	X =  60.822  mm,	Y =   -346.772  mm,	Z =   -269.437  mm,
	W =  90.000 deg,	P =   0.000 deg,	R =   90.000 deg
};
P[82]{
   GP1:
	UF : 0, UT : 6,		CONFIG : 'N U T, 0, 0, 0',
	X =  61.497  mm,	Y =   -348.015  mm,	Z =   -269.167  mm,
	W =  90.000 deg,	P =   0.000 deg,	R =   90.000 deg
};
P[83]{
   GP1:
	UF : 0, UT : 6,		CONFIG : 'N U T, 0, 0, 0',
	X =  62.377  mm,	Y =   -349.588  mm,	Z =   -268.993  mm,
	W =  90.000 deg,	P =   0.000 deg,	R =   90.000 deg
};
P[84]{
   GP1:
	UF : 0, UT : 6,		CONFIG : 'N U T, 0, 0, 0',
	X =  62.802  mm,	Y =   -350.203  mm,	Z =   -269.422  mm,
	W =  90.000 deg,	P =   0.000 deg,	R =   90.000 deg
};
P[85]{
   GP1:
	UF : 0, UT : 6,		CONFIG : 'N U T, 0, 0, 0',
	X =  65.907  mm,	Y =   -355.659  mm,	Z =   -269.143  mm,
	W =  90.000 deg,	P =   0.000 deg,	R =   90.000 deg
};
P[86]{
   GP1:
	UF : 0, UT : 6,		CONFIG : 'N U T, 0, 0, 0',
	X =  66.444  mm,	Y =   -356.602  mm,	Z =   -269.105  mm,
	W =  90.000 deg,	P =   0.000 deg,	R =   90.000 deg
};
P[87]{
   GP1:
	UF : 0, UT : 6,		CONFIG : 'N U T, 0, 0, 0',
	X =  67.551  mm,	Y =   -358.541  mm,	Z =   -269.018  mm,
	W =  90.000 deg,	P =   0.000 deg,	R =   90.000 deg
};
P[88]{
   GP1:
	UF : 0, UT : 6,		CONFIG : 'N U T, 0, 0, 0',
	X =  68.086  mm,	Y =   -359.347  mm,	Z =   -269.445  mm,
	W =  90.000 deg,	P =   0.000 deg,	R =   90.000 deg
};
P[89]{
   GP1:
	UF : 0, UT : 6,		CONFIG : 'N U T, 0, 0, 0',
	X =  68.697  mm,	Y =   -360.426  mm,	Z =   -269.380  mm,
	W =  90.000 deg,	P =   0.000 deg,	R =   90.000 deg
};
P[90]{
   GP1:
	UF : 0, UT : 6,		CONFIG : 'N U T, 0, 0, 0',
	X =  69.791  mm,	Y =   -362.363  mm,	Z =   -269.223  mm,
	W =  90.000 deg,	P =   0.000 deg,	R =   90.000 deg
};
P[91]{
   GP1:
	UF : 0, UT : 6,		CONFIG : 'N U T, 0, 0, 0',
	X =  70.454  mm,	Y =   -363.448  mm,	Z =   -269.452  mm,
	W =  90.000 deg,	P =   0.000 deg,	R =   90.000 deg
};
P[92]{
   GP1:
	UF : 0, UT : 6,		CONFIG : 'N U T, 0, 0, 0',
	X =  71.652  mm,	Y =   -365.531  mm,	Z =   -269.420  mm,
	W =  90.000 deg,	P =   0.000 deg,	R =   90.000 deg
};
P[93]{
   GP1:
	UF : 0, UT : 6,		CONFIG : 'N U T, 0, 0, 0',
	X =  72.017  mm,	Y =   -366.190  mm,	Z =   -269.328  mm,
	W =  90.000 deg,	P =   0.000 deg,	R =   90.000 deg
};
P[94]{
   GP1:
	UF : 0, UT : 6,		CONFIG : 'N U T, 0, 0, 0',
	X =  73.518  mm,	Y =   -368.753  mm,	Z =   -269.459  mm,
	W =  90.000 deg,	P =   0.000 deg,	R =   90.000 deg
};
P[95]{
   GP1:
	UF : 0, UT : 6,		CONFIG : 'N U T, 0, 0, 0',
	X =  74.232  mm,	Y =   -370.046  mm,	Z =   -269.257  mm,
	W =  90.000 deg,	P =   0.000 deg,	R =   90.000 deg
};
P[96]{
   GP1:
	UF : 0, UT : 6,		CONFIG : 'N U T, 0, 0, 0',
	X =  75.118  mm,	Y =   -371.588  mm,	Z =   -269.233  mm,
	W =  90.000 deg,	P =   0.000 deg,	R =   90.000 deg
};
P[97]{
   GP1:
	UF : 0, UT : 6,		CONFIG : 'N U T, 0, 0, 0',
	X =  76.161  mm,	Y =   -373.400  mm,	Z =   -269.214  mm,
	W =  90.000 deg,	P =   0.000 deg,	R =   90.000 deg
};
P[98]{
   GP1:
	UF : 0, UT : 6,		CONFIG : 'N U T, 0, 0, 0',
	X =  76.622  mm,	Y =   -374.139  mm,	Z =   -269.425  mm,
	W =  90.000 deg,	P =   0.000 deg,	R =   90.000 deg
};
P[99]{
   GP1:
	UF : 0, UT : 6,		CONFIG : 'N U T, 0, 0, 0',
	X =  77.809  mm,	Y =   -376.265  mm,	Z =   -269.174  mm,
	W =  90.000 deg,	P =   0.000 deg,	R =   90.000 deg
};
P[100]{
   GP1:
	UF : 0, UT : 6,		CONFIG : 'N U T, 0, 0, 0',
	X =  78.464  mm,	Y =   -377.334  mm,	Z =   -269.401  mm,
	W =  90.000 deg,	P =   0.000 deg,	R =   90.000 deg
};
P[101]{
   GP1:
	UF : 0, UT : 6,		CONFIG : 'N U T, 0, 0, 0',
	X =  78.788  mm,	Y =   -377.936  mm,	Z =   -269.254  mm,
	W =  90.000 deg,	P =   0.000 deg,	R =   90.000 deg
};
P[102]{
   GP1:
	UF : 0, UT : 6,		CONFIG : 'N U T, 0, 0, 0',
	X =  79.817  mm,	Y =   -379.792  mm,	Z =   -268.996  mm,
	W =  90.000 deg,	P =   0.000 deg,	R =   90.000 deg
};
P[103]{
   GP1:
	UF : 0, UT : 6,		CONFIG : 'N U T, 0, 0, 0',
	X =  80.835  mm,	Y =   -381.493  mm,	Z =   -269.218  mm,
	W =  90.000 deg,	P =   0.000 deg,	R =   90.000 deg
};
P[104]{
   GP1:
	UF : 0, UT : 6,		CONFIG : 'N U T, 0, 0, 0',
	X =  81.508  mm,	Y =   -382.632  mm,	Z =   -269.316  mm,
	W =  90.000 deg,	P =   0.000 deg,	R =   90.000 deg
};
P[105]{
   GP1:
	UF : 0, UT : 6,		CONFIG : 'N U T, 0, 0, 0',
	X =  82.678  mm,	Y =   -384.651  mm,	Z =   -269.338  mm,
	W =  90.000 deg,	P =   0.000 deg,	R =   90.000 deg
};
P[106]{
   GP1:
	UF : 0, UT : 6,		CONFIG : 'N U T, 0, 0, 0',
	X =  83.057  mm,	Y =   -385.408  mm,	Z =   -268.979  mm,
	W =  90.000 deg,	P =   0.000 deg,	R =   90.000 deg
};
P[107]{
   GP1:
	UF : 0, UT : 6,		CONFIG : 'N U T, 0, 0, 0',
	X =  83.869  mm,	Y =   -386.793  mm,	Z =   -269.051  mm,
	W =  90.000 deg,	P =   0.000 deg,	R =   90.000 deg
};
P[108]{
   GP1:
	UF : 0, UT : 6,		CONFIG : 'N U T, 0, 0, 0',
	X =  84.504  mm,	Y =   -387.810  mm,	Z =   -269.347  mm,
	W =  90.000 deg,	P =   0.000 deg,	R =   90.000 deg
};
P[109]{
   GP1:
	UF : 0, UT : 6,		CONFIG : 'N U T, 0, 0, 0',
	X =  85.651  mm,	Y =   -389.786  mm,	Z =   -269.386  mm,
	W =  90.000 deg,	P =   0.000 deg,	R =   90.000 deg
};
P[110]{
   GP1:
	UF : 0, UT : 6,		CONFIG : 'N U T, 0, 0, 0',
	X =  86.141  mm,	Y =   -390.741  mm,	Z =   -269.016  mm,
	W =  90.000 deg,	P =   0.000 deg,	R =   90.000 deg
};
P[111]{
   GP1:
	UF : 0, UT : 6,		CONFIG : 'N U T, 0, 0, 0',
	X =  87.192  mm,	Y =   -392.497  mm,	Z =   -269.239  mm,
	W =  90.000 deg,	P =   0.000 deg,	R =   90.000 deg
};
P[112]{
   GP1:
	UF : 0, UT : 6,		CONFIG : 'N U T, 0, 0, 0',
	X =  88.643  mm,	Y =   -394.957  mm,	Z =   -269.426  mm,
	W =  90.000 deg,	P =   0.000 deg,	R =   90.000 deg
};
P[113]{
   GP1:
	UF : 0, UT : 6,		CONFIG : 'N U T, 0, 0, 0',
	X =  89.008  mm,	Y =   -395.619  mm,	Z =   -269.324  mm,
	W =  90.000 deg,	P =   0.000 deg,	R =   90.000 deg
};
P[114]{
   GP1:
	UF : 0, UT : 6,		CONFIG : 'N U T, 0, 0, 0',
	X =  89.567  mm,	Y =   -396.633  mm,	Z =   -269.159  mm,
	W =  90.000 deg,	P =   0.000 deg,	R =   90.000 deg
};
P[115]{
   GP1:
	UF : 0, UT : 6,		CONFIG : 'N U T, 0, 0, 0',
	X =  89.934  mm,	Y =   -397.204  mm,	Z =   -269.389  mm,
	W =  90.000 deg,	P =   0.000 deg,	R =   90.000 deg
};
P[116]{
   GP1:
	UF : 0, UT : 6,		CONFIG : 'N U T, 0, 0, 0',
	X =  90.802  mm,	Y =   -398.817  mm,	Z =   -269.000  mm,
	W =  90.000 deg,	P =   0.000 deg,	R =   90.000 deg
};
P[117]{
   GP1:
	UF : 0, UT : 6,		CONFIG : 'N U T, 0, 0, 0',
	X =  91.673  mm,	Y =   -400.288  mm,	Z =   -269.133  mm,
	W =  90.000 deg,	P =   0.000 deg,	R =   90.000 deg
};
P[118]{
   GP1:
	UF : 0, UT : 6,		CONFIG : 'N U T, 0, 0, 0',
	X =  92.270  mm,	Y =   -401.280  mm,	Z =   -269.279  mm,
	W =  90.000 deg,	P =   0.000 deg,	R =   90.000 deg
};
P[119]{
   GP1:
	UF : 0, UT : 6,		CONFIG : 'N U T, 0, 0, 0',
	X =  92.609  mm,	Y =   -401.953  mm,	Z =   -268.976  mm,
	W =  90.000 deg,	P =   0.000 deg,	R =   90.000 deg
};
P[120]{
   GP1:
	UF : 0, UT : 6,		CONFIG : 'N U T, 0, 0, 0',
	X =  93.263  mm,	Y =   -402.984  mm,	Z =   -269.335  mm,
	W =  90.000 deg,	P =   0.000 deg,	R =   90.000 deg
};
P[121]{
   GP1:
	UF : 0, UT : 6,		CONFIG : 'N U T, 0, 0, 0',
	X =  94.215  mm,	Y =   -404.733  mm,	Z =   -268.981  mm,
	W =  90.000 deg,	P =   0.000 deg,	R =   90.000 deg
};
P[122]{
   GP1:
	UF : 0, UT : 6,		CONFIG : 'N U T, 0, 0, 0',
	X =  94.663  mm,	Y =   -405.406  mm,	Z =   -269.352  mm,
	W =  90.000 deg,	P =   0.000 deg,	R =   90.000 deg
};
P[123]{
   GP1:
	UF : 0, UT : 6,		CONFIG : 'N U T, 0, 0, 0',
	X =  95.233  mm,	Y =   -406.415  mm,	Z =   -269.271  mm,
	W =  90.000 deg,	P =   0.000 deg,	R =   90.000 deg
};
P[124]{
   GP1:
	UF : 0, UT : 6,		CONFIG : 'N U T, 0, 0, 0',
	X =  95.633  mm,	Y =   -407.055  mm,	Z =   -269.454  mm,
	W =  90.000 deg,	P =   0.000 deg,	R =   90.000 deg
};
P[125]{
   GP1:
	UF : 0, UT : 6,		CONFIG : 'N U T, 0, 0, 0',
	X =  96.047  mm,	Y =   -407.781  mm,	Z =   -269.422  mm,
	W =  90.000 deg,	P =   0.000 deg,	R =   90.000 deg
};
P[126]{
   GP1:
	UF : 0, UT : 6,		CONFIG : 'N U T, 0, 0, 0',
	X =  96.838  mm,	Y =   -409.146  mm,	Z =   -269.439  mm,
	W =  90.000 deg,	P =   0.000 deg,	R =   90.000 deg
};
P[127]{
   GP1:
	UF : 0, UT : 6,		CONFIG : 'N U T, 0, 0, 0',
	X =  97.336  mm,	Y =   -410.021  mm,	Z =   -269.398  mm,
	W =  90.000 deg,	P =   0.000 deg,	R =   90.000 deg
};
P[128]{
   GP1:
	UF : 0, UT : 6,		CONFIG : 'N U T, 0, 0, 0',
	X =  100.649  mm,	Y =   -415.788  mm,	Z =   -269.295  mm,
	W =  90.000 deg,	P =   0.000 deg,	R =   90.000 deg
};
P[129]{
   GP1:
	UF : 0, UT : 6,		CONFIG : 'N U T, 0, 0, 0',
	X =  101.557  mm,	Y =   -417.366  mm,	Z =   -269.280  mm,
	W =  90.000 deg,	P =   0.000 deg,	R =   90.000 deg
};
P[130]{
   GP1:
	UF : 0, UT : 6,		CONFIG : 'N U T, 0, 0, 0',
	X =  102.068  mm,	Y =   -418.216  mm,	Z =   -269.399  mm,
	W =  90.000 deg,	P =   0.000 deg,	R =   90.000 deg
};
P[131]{
   GP1:
	UF : 0, UT : 6,		CONFIG : 'N U T, 0, 0, 0',
	X =  102.519  mm,	Y =   -419.075  mm,	Z =   -269.120  mm,
	W =  90.000 deg,	P =   0.000 deg,	R =   90.000 deg
};
P[132]{
   GP1:
	UF : 0, UT : 6,		CONFIG : 'N U T, 0, 0, 0',
	X =  102.875  mm,	Y =   -419.712  mm,	Z =   -269.046  mm,
	W =  90.000 deg,	P =   0.000 deg,	R =   90.000 deg
};
P[133]{
   GP1:
	UF : 0, UT : 6,		CONFIG : 'N U T, 0, 0, 0',
	X =  103.510  mm,	Y =   -420.772  mm,	Z =   -269.198  mm,
	W =  90.000 deg,	P =   0.000 deg,	R =   90.000 deg
};
P[134]{
   GP1:
	UF : 0, UT : 6,		CONFIG : 'N U T, 0, 0, 0',
	X =  104.292  mm,	Y =   -422.113  mm,	Z =   -269.234  mm,
	W =  90.000 deg,	P =   0.000 deg,	R =   90.000 deg
};
P[135]{
   GP1:
	UF : 0, UT : 6,		CONFIG : 'N U T, 0, 0, 0',
	X =  104.762  mm,	Y =   -422.880  mm,	Z =   -269.407  mm,
	W =  90.000 deg,	P =   0.000 deg,	R =   90.000 deg
};
P[136]{
   GP1:
	UF : 0, UT : 6,		CONFIG : 'N U T, 0, 0, 0',
	X =  105.548  mm,	Y =   -424.257  mm,	Z =   -269.352  mm,
	W =  90.000 deg,	P =   0.000 deg,	R =   90.000 deg
};
P[137]{
   GP1:
	UF : 0, UT : 6,		CONFIG : 'N U T, 0, 0, 0',
	X =  106.528  mm,	Y =   -425.936  mm,	Z =   -269.416  mm,
	W =  90.000 deg,	P =   0.000 deg,	R =   90.000 deg
};
P[138]{
   GP1:
	UF : 0, UT : 6,		CONFIG : 'N U T, 0, 0, 0',
	X =  107.193  mm,	Y =   -427.150  mm,	Z =   -269.199  mm,
	W =  90.000 deg,	P =   0.000 deg,	R =   90.000 deg
};
P[139]{
   GP1:
	UF : 0, UT : 6,		CONFIG : 'N U T, 0, 0, 0',
	X =  108.073  mm,	Y =   -428.628  mm,	Z =   -269.361  mm,
	W =  90.000 deg,	P =   0.000 deg,	R =   90.000 deg
};
P[140]{
   GP1:
	UF : 0, UT : 6,		CONFIG : 'N U T, 0, 0, 0',
	X =  108.634  mm,	Y =   -429.629  mm,	Z =   -269.255  mm,
	W =  90.000 deg,	P =   0.000 deg,	R =   90.000 deg
};
P[141]{
   GP1:
	UF : 0, UT : 6,		CONFIG : 'N U T, 0, 0, 0',
	X =  109.762  mm,	Y =   -431.647  mm,	Z =   -269.028  mm,
	W =  90.000 deg,	P =   0.000 deg,	R =   90.000 deg
};
P[142]{
   GP1:
	UF : 0, UT : 6,		CONFIG : 'N U T, 0, 0, 0',
	X =  110.780  mm,	Y =   -433.376  mm,	Z =   -269.148  mm,
	W =  90.000 deg,	P =   0.000 deg,	R =   90.000 deg
};
P[143]{
   GP1:
	UF : 0, UT : 6,		CONFIG : 'N U T, 0, 0, 0',
	X =  112.089  mm,	Y =   -435.605  mm,	Z =   -269.286  mm,
	W =  90.000 deg,	P =   0.000 deg,	R =   90.000 deg
};
P[144]{
   GP1:
	UF : 0, UT : 6,		CONFIG : 'N U T, 0, 0, 0',
	X =  112.688  mm,	Y =   -436.601  mm,	Z =   -269.430  mm,
	W =  90.000 deg,	P =   0.000 deg,	R =   90.000 deg
};
P[145]{
   GP1:
	UF : 0, UT : 6,		CONFIG : 'N U T, 0, 0, 0',
	X =  113.248  mm,	Y =   -437.579  mm,	Z =   -269.400  mm,
	W =  90.000 deg,	P =   0.000 deg,	R =   90.000 deg
};
P[146]{
   GP1:
	UF : 0, UT : 6,		CONFIG : 'N U T, 0, 0, 0',
	X =  115.422  mm,	Y =   -441.341  mm,	Z =   -269.410  mm,
	W =  90.000 deg,	P =   0.000 deg,	R =   90.000 deg
};
P[147]{
   GP1:
	UF : 0, UT : 6,		CONFIG : 'N U T, 0, 0, 0',
	X =  116.395  mm,	Y =   -443.103  mm,	Z =   -269.137  mm,
	W =  90.000 deg,	P =   0.000 deg,	R =   90.000 deg
};
P[148]{
   GP1:
	UF : 0, UT : 6,		CONFIG : 'N U T, 0, 0, 0',
	X =  116.899  mm,	Y =   -443.894  mm,	Z =   -269.431  mm,
	W =  90.000 deg,	P =   0.000 deg,	R =   90.000 deg
};
P[149]{
   GP1:
	UF : 0, UT : 6,		CONFIG : 'N U T, 0, 0, 0',
	X =  117.215  mm,	Y =   -444.562  mm,	Z =   -269.000  mm,
	W =  90.000 deg,	P =   0.000 deg,	R =   90.000 deg
};
P[150]{
   GP1:
	UF : 0, UT : 6,		CONFIG : 'N U T, 0, 0, 0',
	X =  119.568  mm,	Y =   -448.558  mm,	Z =   -269.287  mm,
	W =  90.000 deg,	P =   0.000 deg,	R =   90.000 deg
};
P[151]{
   GP1:
	UF : 0, UT : 6,		CONFIG : 'N U T, 0, 0, 0',
	X =  120.224  mm,	Y =   -449.780  mm,	Z =   -268.978  mm,
	W =  90.000 deg,	P =   0.000 deg,	R =   90.000 deg
};
P[152]{
   GP1:
	UF : 0, UT : 6,		CONFIG : 'N U T, 0, 0, 0',
	X =  120.522  mm,	Y =   -450.161  mm,	Z =   -269.456  mm,
	W =  90.000 deg,	P =   0.000 deg,	R =   90.000 deg
};
P[153]{
   GP1:
	UF : 0, UT : 6,		CONFIG : 'N U T, 0, 0, 0',
	X =  121.028  mm,	Y =   -451.052  mm,	Z =   -269.408  mm,
	W =  90.000 deg,	P =   0.000 deg,	R =   90.000 deg
};
P[154]{
   GP1:
	UF : 0, UT : 6,		CONFIG : 'N U T, 0, 0, 0',
	X =  121.776  mm,	Y =   -452.357  mm,	Z =   -269.371  mm,
	W =  90.000 deg,	P =   0.000 deg,	R =   90.000 deg
};
P[155]{
   GP1:
	UF : 0, UT : 6,		CONFIG : 'N U T, 0, 0, 0',
	X =  122.156  mm,	Y =   -453.037  mm,	Z =   -269.292  mm,
	W =  90.000 deg,	P =   0.000 deg,	R =   90.000 deg
};
P[156]{
   GP1:
	UF : 0, UT : 6,		CONFIG : 'N U T, 0, 0, 0',
	X =  124.148  mm,	Y =   -456.445  mm,	Z =   -269.440  mm,
	W =  90.000 deg,	P =   0.000 deg,	R =   90.000 deg
};
P[157]{
   GP1:
	UF : 0, UT : 6,		CONFIG : 'N U T, 0, 0, 0',
	X =  124.997  mm,	Y =   -457.915  mm,	Z =   -269.440  mm,
	W =  90.000 deg,	P =   0.000 deg,	R =   90.000 deg
};
P[158]{
   GP1:
	UF : 0, UT : 6,		CONFIG : 'N U T, 0, 0, 0',
	X =  125.612  mm,	Y =   -459.081  mm,	Z =   -269.087  mm,
	W =  90.000 deg,	P =   0.000 deg,	R =   90.000 deg
};
P[159]{
   GP1:
	UF : 0, UT : 6,		CONFIG : 'N U T, 0, 0, 0',
	X =  128.158  mm,	Y =   -463.507  mm,	Z =   -269.027  mm,
	W =  90.000 deg,	P =   0.000 deg,	R =   90.000 deg
};
P[160]{
   GP1:
	UF : 0, UT : 6,		CONFIG : 'N U T, 0, 0, 0',
	X =  128.749  mm,	Y =   -464.531  mm,	Z =   -269.030  mm,
	W =  90.000 deg,	P =   0.000 deg,	R =   90.000 deg
};
P[161]{
   GP1:
	UF : 0, UT : 6,		CONFIG : 'N U T, 0, 0, 0',
	X =  129.241  mm,	Y =   -465.284  mm,	Z =   -269.376  mm,
	W =  90.000 deg,	P =   0.000 deg,	R =   90.000 deg
};
P[162]{
   GP1:
	UF : 0, UT : 6,		CONFIG : 'N U T, 0, 0, 0',
	X =  130.318  mm,	Y =   -467.144  mm,	Z =   -269.397  mm,
	W =  90.000 deg,	P =   0.000 deg,	R =   90.000 deg
};
P[163]{
   GP1:
	UF : 0, UT : 6,		CONFIG : 'N U T, 0, 0, 0',
	X =  130.586  mm,	Y =   -467.686  mm,	Z =   -269.122  mm,
	W =  90.000 deg,	P =   0.000 deg,	R =   90.000 deg
};
P[164]{
   GP1:
	UF : 0, UT : 6,		CONFIG : 'N U T, 0, 0, 0',
	X =  131.578  mm,	Y =   -469.327  mm,	Z =   -269.393  mm,
	W =  90.000 deg,	P =   0.000 deg,	R =   90.000 deg
};
P[165]{
   GP1:
	UF : 0, UT : 6,		CONFIG : 'N U T, 0, 0, 0',
	X =  132.526  mm,	Y =   -470.972  mm,	Z =   -269.383  mm,
	W =  90.000 deg,	P =   0.000 deg,	R =   90.000 deg
};
P[166]{
   GP1:
	UF : 0, UT : 6,		CONFIG : 'N U T, 0, 0, 0',
	X =  132.867  mm,	Y =   -471.637  mm,	Z =   -269.117  mm,
	W =  90.000 deg,	P =   0.000 deg,	R =   90.000 deg
};
P[167]{
   GP1:
	UF : 0, UT : 6,		CONFIG : 'N U T, 0, 0, 0',
	X =  133.655  mm,	Y =   -473.001  mm,	Z =   -269.117  mm,
	W =  90.000 deg,	P =   0.000 deg,	R =   90.000 deg
};
P[168]{
   GP1:
	UF : 0, UT : 6,		CONFIG : 'N U T, 0, 0, 0',
	X =  134.696  mm,	Y =   -474.789  mm,	Z =   -269.170  mm,
	W =  90.000 deg,	P =   0.000 deg,	R =   90.000 deg
};
P[169]{
   GP1:
	UF : 0, UT : 6,		CONFIG : 'N U T, 0, 0, 0',
	X =  135.766  mm,	Y =   -476.584  mm,	Z =   -269.382  mm,
	W =  90.000 deg,	P =   0.000 deg,	R =   90.000 deg
};
P[170]{
   GP1:
	UF : 0, UT : 6,		CONFIG : 'N U T, 0, 0, 0',
	X =  136.419  mm,	Y =   -477.710  mm,	Z =   -269.402  mm,
	W =  90.000 deg,	P =   0.000 deg,	R =   90.000 deg
};
P[171]{
   GP1:
	UF : 0, UT : 6,		CONFIG : 'N U T, 0, 0, 0',
	X =  136.740  mm,	Y =   -478.303  mm,	Z =   -269.264  mm,
	W =  90.000 deg,	P =   0.000 deg,	R =   90.000 deg
};
P[172]{
   GP1:
	UF : 0, UT : 6,		CONFIG : 'N U T, 0, 0, 0',
	X =  137.648  mm,	Y =   -479.881  mm,	Z =   -269.246  mm,
	W =  90.000 deg,	P =   0.000 deg,	R =   90.000 deg
};
P[173]{
   GP1:
	UF : 0, UT : 6,		CONFIG : 'N U T, 0, 0, 0',
	X =  138.018  mm,	Y =   -480.494  mm,	Z =   -269.352  mm,
	W =  90.000 deg,	P =   0.000 deg,	R =   90.000 deg
};
P[174]{
   GP1:
	UF : 0, UT : 6,		CONFIG : 'N U T, 0, 0, 0',
	X =  138.408  mm,	Y =   -481.170  mm,	Z =   -269.340  mm,
	W =  90.000 deg,	P =   0.000 deg,	R =   90.000 deg
};
P[175]{
   GP1:
	UF : 0, UT : 6,		CONFIG : 'N U T, 0, 0, 0',
	X =  138.842  mm,	Y =   -481.910  mm,	Z =   -269.379  mm,
	W =  90.000 deg,	P =   0.000 deg,	R =   90.000 deg
};
P[176]{
   GP1:
	UF : 0, UT : 6,		CONFIG : 'N U T, 0, 0, 0',
	X =  140.130  mm,	Y =   -484.202  mm,	Z =   -269.165  mm,
	W =  90.000 deg,	P =   0.000 deg,	R =   90.000 deg
};
P[177]{
   GP1:
	UF : 0, UT : 6,		CONFIG : 'N U T, 0, 0, 0',
	X =  140.790  mm,	Y =   -485.264  mm,	Z =   -269.453  mm,
	W =  90.000 deg,	P =   0.000 deg,	R =   90.000 deg
};
P[178]{
   GP1:
	UF : 0, UT : 6,		CONFIG : 'N U T, 0, 0, 0',
	X =  141.212  mm,	Y =   -486.021  mm,	Z =   -269.362  mm,
	W =  90.000 deg,	P =   0.000 deg,	R =   90.000 deg
};
P[179]{
   GP1:
	UF : 0, UT : 6,		CONFIG : 'N U T, 0, 0, 0',
	X =  141.744  mm,	Y =   -486.945  mm,	Z =   -269.355  mm,
	W =  90.000 deg,	P =   0.000 deg,	R =   90.000 deg
};
P[180]{
   GP1:
	UF : 0, UT : 6,		CONFIG : 'N U T, 0, 0, 0',
	X =  142.350  mm,	Y =   -488.009  mm,	Z =   -269.302  mm,
	W =  90.000 deg,	P =   0.000 deg,	R =   90.000 deg
};
P[181]{
   GP1:
	UF : 0, UT : 6,		CONFIG : 'N U T, 0, 0, 0',
	X =  142.817  mm,	Y =   -488.781  mm,	Z =   -269.437  mm,
	W =  90.000 deg,	P =   0.000 deg,	R =   90.000 deg
};
P[182]{
   GP1:
	UF : 0, UT : 6,		CONFIG : 'N U T, 0, 0, 0',
	X =  143.151  mm,	Y =   -489.474  mm,	Z =   -269.027  mm,
	W =  90.000 deg,	P =   0.000 deg,	R =   90.000 deg
};
P[183]{
   GP1:
	UF : 0, UT : 6,		CONFIG : 'N U T, 0, 0, 0',
	X =  144.297  mm,	Y =   -491.429  mm,	Z =   -269.133  mm,
	W =  90.000 deg,	P =   0.000 deg,	R =   90.000 deg
};
P[184]{
   GP1:
	UF : 0, UT : 6,		CONFIG : 'N U T, 0, 0, 0',
	X =  144.808  mm,	Y =   -492.245  mm,	Z =   -269.373  mm,
	W =  90.000 deg,	P =   0.000 deg,	R =   90.000 deg
};
P[185]{
   GP1:
	UF : 0, UT : 6,		CONFIG : 'N U T, 0, 0, 0',
	X =  145.561  mm,	Y =   -493.548  mm,	Z =   -269.383  mm,
	W =  90.000 deg,	P =   0.000 deg,	R =   90.000 deg
};
P[186]{
   GP1:
	UF : 0, UT : 6,		CONFIG : 'N U T, 0, 0, 0',
	X =  146.862  mm,	Y =   -495.883  mm,	Z =   -269.093  mm,
	W =  90.000 deg,	P =   0.000 deg,	R =   90.000 deg
};
P[187]{
   GP1:
	UF : 0, UT : 6,		CONFIG : 'N U T, 0, 0, 0',
	X =  147.416  mm,	Y =   -496.821  mm,	Z =   -269.162  mm,
	W =  90.000 deg,	P =   0.000 deg,	R =   90.000 deg
};
P[188]{
   GP1:
	UF : 0, UT : 6,		CONFIG : 'N U T, 0, 0, 0',
	X =  147.915  mm,	Y =   -497.610  mm,	Z =   -269.436  mm,
	W =  90.000 deg,	P =   0.000 deg,	R =   90.000 deg
};
P[189]{
   GP1:
	UF : 0, UT : 6,		CONFIG : 'N U T, 0, 0, 0',
	X =  148.320  mm,	Y =   -498.396  mm,	Z =   -269.133  mm,
	W =  90.000 deg,	P =   0.000 deg,	R =   90.000 deg
};
P[190]{
   GP1:
	UF : 0, UT : 6,		CONFIG : 'N U T, 0, 0, 0',
	X =  149.677  mm,	Y =   -500.726  mm,	Z =   -269.202  mm,
	W =  90.000 deg,	P =   0.000 deg,	R =   90.000 deg
};
P[191]{
   GP1:
	UF : 0, UT : 6,		CONFIG : 'N U T, 0, 0, 0',
	X =  151.048  mm,	Y =   -503.071  mm,	Z =   -269.312  mm,
	W =  90.000 deg,	P =   0.000 deg,	R =   90.000 deg
};
P[192]{
   GP1:
	UF : 0, UT : 6,		CONFIG : 'N U T, 0, 0, 0',
	X =  151.586  mm,	Y =   -504.006  mm,	Z =   -269.295  mm,
	W =  90.000 deg,	P =   0.000 deg,	R =   90.000 deg
};
P[193]{
   GP1:
	UF : 0, UT : 6,		CONFIG : 'N U T, 0, 0, 0',
	X =  152.102  mm,	Y =   -504.974  mm,	Z =   -269.037  mm,
	W =  90.000 deg,	P =   0.000 deg,	R =   90.000 deg
};
P[194]{
   GP1:
	UF : 0, UT : 6,		CONFIG : 'N U T, 0, 0, 0',
	X =  153.212  mm,	Y =   -506.878  mm,	Z =   -269.100  mm,
	W =  90.000 deg,	P =   0.000 deg,	R =   90.000 deg
};
P[195]{
   GP1:
	UF : 0, UT : 6,		CONFIG : 'N U T, 0, 0, 0',
	X =  153.818  mm,	Y =   -507.871  mm,	Z =   -269.303  mm,
	W =  90.000 deg,	P =   0.000 deg,	R =   90.000 deg
};
P[196]{
   GP1:
	UF : 0, UT : 6,		CONFIG : 'N U T, 0, 0, 0',
	X =  154.676  mm,	Y =   -509.415  mm,	Z =   -269.092  mm,
	W =  90.000 deg,	P =   0.000 deg,	R =   90.000 deg
};
P[197]{
   GP1:
	UF : 0, UT : 6,		CONFIG : 'N U T, 0, 0, 0',
	X =  155.617  mm,	Y =   -511.066  mm,	Z =   -269.019  mm,
	W =  90.000 deg,	P =   0.000 deg,	R =   90.000 deg
};
P[198]{
   GP1:
	UF : 0, UT : 6,		CONFIG : 'N U T, 0, 0, 0',
	X =  158.474  mm,	Y =   -515.945  mm,	Z =   -269.263  mm,
	W =  90.000 deg,	P =   0.000 deg,	R =   90.000 deg
};
P[199]{
   GP1:
	UF : 0, UT : 6,		CONFIG : 'N U T, 0, 0, 0',
	X =  158.853  mm,	Y =   -516.596  mm,	Z =   -269.285  mm,
	W =  90.000 deg,	P =   0.000 deg,	R =   90.000 deg
};
P[200]{
   GP1:
	UF : 0, UT : 6,		CONFIG : 'N U T, 0, 0, 0',
	X =  159.441  mm,	Y =   -517.703  mm,	Z =   -268.966  mm,
	W =  90.000 deg,	P =   0.000 deg,	R =   90.000 deg
};
P[201]{
   GP1:
	UF : 0, UT : 6,		CONFIG : 'N U T, 0, 0, 0',
	X =  161.036  mm,	Y =   -520.410  mm,	Z =   -269.167  mm,
	W =  90.000 deg,	P =   0.000 deg,	R =   90.000 deg
};
P[202]{
   GP1:
	UF : 0, UT : 6,		CONFIG : 'N U T, 0, 0, 0',
	X =  161.382  mm,	Y =   -521.000  mm,	Z =   -269.199  mm,
	W =  90.000 deg,	P =   0.000 deg,	R =   90.000 deg
};
P[203]{
   GP1:
	UF : 0, UT : 6,		CONFIG : 'N U T, 0, 0, 0',
	X =  162.364  mm,	Y =   -522.664  mm,	Z =   -269.330  mm,
	W =  90.000 deg,	P =   0.000 deg,	R =   90.000 deg
};
P[204]{
   GP1:
	UF : 0, UT : 6,		CONFIG : 'N U T, 0, 0, 0',
	X =  164.500  mm,	Y =   -526.438  mm,	Z =   -269.066  mm,
	W =  90.000 deg,	P =   0.000 deg,	R =   90.000 deg
};
P[205]{
   GP1:
	UF : 0, UT : 6,		CONFIG : 'N U T, 0, 0, 0',
	X =  164.852  mm,	Y =   -527.016  mm,	Z =   -269.170  mm,
	W =  90.000 deg,	P =   0.000 deg,	R =   90.000 deg
};
P[206]{
   GP1:
	UF : 0, UT : 6,		CONFIG : 'N U T, 0, 0, 0',
	X =  165.400  mm,	Y =   -527.931  mm,	Z =   -269.296  mm,
	W =  90.000 deg,	P =   0.000 deg,	R =   90.000 deg
};
P[207]{
   GP1:
	UF : 0, UT : 6,		CONFIG : 'N U T, 0, 0, 0',
	X =  165.758  mm,	Y =   -528.605  mm,	Z =   -269.109  mm,
	W =  90.000 deg,	P =   0.000 deg,	R =   90.000 deg
};
P[208]{
   GP1:
	UF : 0, UT : 6,		CONFIG : 'N U T, 0, 0, 0',
	X =  167.042  mm,	Y =   -530.004  mm,	Z =   -269.068  mm,
	W =  90.000 deg,	P =   0.000 deg,	R =   90.000 deg
};
P[209]{
   GP1:
	UF : 0, UT : 6,		CONFIG : 'N U T, 0, 0, 0',
	X =  168.359  mm,	Y =   -530.573  mm,	Z =   -269.374  mm,
	W =  90.000 deg,	P =   0.000 deg,	R =   90.000 deg
};
P[210]{
   GP1:
	UF : 0, UT : 6,		CONFIG : 'N U T, 0, 0, 0',
	X =  168.920  mm,	Y =   -530.716  mm,	Z =   -269.021  mm,
	W =  90.000 deg,	P =   0.000 deg,	R =   90.000 deg
};
P[211]{
   GP1:
	UF : 0, UT : 6,		CONFIG : 'N U T, 0, 0, 0',
	X =  170.432  mm,	Y =   -530.619  mm,	Z =   -269.093  mm,
	W =  90.000 deg,	P =   0.000 deg,	R =   90.000 deg
};
P[212]{
   GP1:
	UF : 0, UT : 6,		CONFIG : 'N U T, 0, 0, 0',
	X =  171.510  mm,	Y =   -530.115  mm,	Z =   -269.355  mm,
	W =  90.000 deg,	P =   0.000 deg,	R =   90.000 deg
};
P[213]{
   GP1:
	UF : 0, UT : 6,		CONFIG : 'N U T, 0, 0, 0',
	X =  172.742  mm,	Y =   -529.395  mm,	Z =   -269.414  mm,
	W =  90.000 deg,	P =   0.000 deg,	R =   90.000 deg
};
P[214]{
   GP1:
	UF : 0, UT : 6,		CONFIG : 'N U T, 0, 0, 0',
	X =  173.815  mm,	Y =   -528.835  mm,	Z =   -269.049  mm,
	W =  90.000 deg,	P =   0.000 deg,	R =   90.000 deg
};
P[215]{
   GP1:
	UF : 0, UT : 6,		CONFIG : 'N U T, 0, 0, 0',
	X =  174.508  mm,	Y =   -528.392  mm,	Z =   -269.310  mm,
	W =  90.000 deg,	P =   0.000 deg,	R =   90.000 deg
};
P[216]{
   GP1:
	UF : 0, UT : 6,		CONFIG : 'N U T, 0, 0, 0',
	X =  176.431  mm,	Y =   -527.258  mm,	Z =   -269.458  mm,
	W =  90.000 deg,	P =   0.000 deg,	R =   90.000 deg
};
P[217]{
   GP1:
	UF : 0, UT : 6,		CONFIG : 'N U T, 0, 0, 0',
	X =  177.653  mm,	Y =   -526.579  mm,	Z =   -269.291  mm,
	W =  90.000 deg,	P =   0.000 deg,	R =   90.000 deg
};
P[218]{
   GP1:
	UF : 0, UT : 6,		CONFIG : 'N U T, 0, 0, 0',
	X =  180.438  mm,	Y =   -524.968  mm,	Z =   -269.312  mm,
	W =  90.000 deg,	P =   0.000 deg,	R =   90.000 deg
};
P[219]{
   GP1:
	UF : 0, UT : 6,		CONFIG : 'N U T, 0, 0, 0',
	X =  181.666  mm,	Y =   -524.240  mm,	Z =   -269.427  mm,
	W =  90.000 deg,	P =   0.000 deg,	R =   90.000 deg
};
P[220]{
   GP1:
	UF : 0, UT : 6,		CONFIG : 'N U T, 0, 0, 0',
	X =  182.795  mm,	Y =   -523.662  mm,	Z =   -268.977  mm,
	W =  90.000 deg,	P =   0.000 deg,	R =   90.000 deg
};
P[221]{
   GP1:
	UF : 0, UT : 6,		CONFIG : 'N U T, 0, 0, 0',
	X =  183.884  mm,	Y =   -522.956  mm,	Z =   -269.447  mm,
	W =  90.000 deg,	P =   0.000 deg,	R =   90.000 deg
};
P[222]{
   GP1:
	UF : 0, UT : 6,		CONFIG : 'N U T, 0, 0, 0',
	X =  186.807  mm,	Y =   -521.268  mm,	Z =   -269.445  mm,
	W =  90.000 deg,	P =   0.000 deg,	R =   90.000 deg
};
P[223]{
   GP1:
	UF : 0, UT : 6,		CONFIG : 'N U T, 0, 0, 0',
	X =  187.667  mm,	Y =   -520.785  mm,	Z =   -269.365  mm,
	W =  90.000 deg,	P =   0.000 deg,	R =   90.000 deg
};
P[224]{
   GP1:
	UF : 0, UT : 6,		CONFIG : 'N U T, 0, 0, 0',
	X =  188.487  mm,	Y =   -520.349  mm,	Z =   -269.132  mm,
	W =  90.000 deg,	P =   0.000 deg,	R =   90.000 deg
};
P[225]{
   GP1:
	UF : 0, UT : 6,		CONFIG : 'N U T, 0, 0, 0',
	X =  190.660  mm,	Y =   -519.066  mm,	Z =   -269.308  mm,
	W =  90.000 deg,	P =   0.000 deg,	R =   90.000 deg
};
P[226]{
   GP1:
	UF : 0, UT : 6,		CONFIG : 'N U T, 0, 0, 0',
	X =  191.705  mm,	Y =   -518.443  mm,	Z =   -269.427  mm,
	W =  90.000 deg,	P =   0.000 deg,	R =   90.000 deg
};
P[227]{
   GP1:
	UF : 0, UT : 6,		CONFIG : 'N U T, 0, 0, 0',
	X =  193.802  mm,	Y =   -517.252  mm,	Z =   -269.307  mm,
	W =  90.000 deg,	P =   0.000 deg,	R =   90.000 deg
};
P[228]{
   GP1:
	UF : 0, UT : 6,		CONFIG : 'N U T, 0, 0, 0',
	X =  195.098  mm,	Y =   -516.521  mm,	Z =   -269.207  mm,
	W =  90.000 deg,	P =   0.000 deg,	R =   90.000 deg
};
P[229]{
   GP1:
	UF : 0, UT : 6,		CONFIG : 'N U T, 0, 0, 0',
	X =  196.970  mm,	Y =   -515.453  mm,	Z =   -269.120  mm,
	W =  90.000 deg,	P =   0.000 deg,	R =   90.000 deg
};
P[230]{
   GP1:
	UF : 0, UT : 6,		CONFIG : 'N U T, 0, 0, 0',
	X =  198.063  mm,	Y =   -514.796  mm,	Z =   -269.281  mm,
	W =  90.000 deg,	P =   0.000 deg,	R =   90.000 deg
};
P[231]{
   GP1:
	UF : 0, UT : 6,		CONFIG : 'N U T, 0, 0, 0',
	X =  199.597  mm,	Y =   -513.914  mm,	Z =   -269.257  mm,
	W =  90.000 deg,	P =   0.000 deg,	R =   90.000 deg
};
P[232]{
   GP1:
	UF : 0, UT : 6,		CONFIG : 'N U T, 0, 0, 0',
	X =  200.332  mm,	Y =   -513.526  mm,	Z =   -269.034  mm,
	W =  90.000 deg,	P =   0.000 deg,	R =   90.000 deg
};
P[233]{
   GP1:
	UF : 0, UT : 6,		CONFIG : 'N U T, 0, 0, 0',
	X =  200.961  mm,	Y =   -513.149  mm,	Z =   -269.120  mm,
	W =  90.000 deg,	P =   0.000 deg,	R =   90.000 deg
};
P[234]{
   GP1:
	UF : 0, UT : 6,		CONFIG : 'N U T, 0, 0, 0',
	X =  202.369  mm,	Y =   -512.336  mm,	Z =   -269.119  mm,
	W =  90.000 deg,	P =   0.000 deg,	R =   90.000 deg
};
P[235]{
   GP1:
	UF : 0, UT : 6,		CONFIG : 'N U T, 0, 0, 0',
	X =  203.269  mm,	Y =   -511.812  mm,	Z =   -269.145  mm,
	W =  90.000 deg,	P =   0.000 deg,	R =   90.000 deg
};
P[236]{
   GP1:
	UF : 0, UT : 6,		CONFIG : 'N U T, 0, 0, 0',
	X =  204.822  mm,	Y =   -510.925  mm,	Z =   -269.085  mm,
	W =  90.000 deg,	P =   0.000 deg,	R =   90.000 deg
};
P[237]{
   GP1:
	UF : 0, UT : 6,		CONFIG : 'N U T, 0, 0, 0',
	X =  205.609  mm,	Y =   -510.433  mm,	Z =   -269.316  mm,
	W =  90.000 deg,	P =   0.000 deg,	R =   90.000 deg
};
P[238]{
   GP1:
	UF : 0, UT : 6,		CONFIG : 'N U T, 0, 0, 0',
	X =  207.390  mm,	Y =   -509.422  mm,	Z =   -269.208  mm,
	W =  90.000 deg,	P =   0.000 deg,	R =   90.000 deg
};
P[239]{
   GP1:
	UF : 0, UT : 6,		CONFIG : 'N U T, 0, 0, 0',
	X =  208.873  mm,	Y =   -508.548  mm,	Z =   -269.321  mm,
	W =  90.000 deg,	P =   0.000 deg,	R =   90.000 deg
};
P[240]{
   GP1:
	UF : 0, UT : 6,		CONFIG : 'N U T, 0, 0, 0',
	X =  209.702  mm,	Y =   -508.104  mm,	Z =   -269.103  mm,
	W =  90.000 deg,	P =   0.000 deg,	R =   90.000 deg
};
P[241]{
   GP1:
	UF : 0, UT : 6,		CONFIG : 'N U T, 0, 0, 0',
	X =  210.796  mm,	Y =   -507.435  mm,	Z =   -269.336  mm,
	W =  90.000 deg,	P =   0.000 deg,	R =   90.000 deg
};
P[242]{
   GP1:
	UF : 0, UT : 6,		CONFIG : 'N U T, 0, 0, 0',
	X =  213.704  mm,	Y =   -505.760  mm,	Z =   -269.309  mm,
	W =  90.000 deg,	P =   0.000 deg,	R =   90.000 deg
};
P[243]{
   GP1:
	UF : 0, UT : 6,		CONFIG : 'N U T, 0, 0, 0',
	X =  214.582  mm,	Y =   -505.242  mm,	Z =   -269.381  mm,
	W =  90.000 deg,	P =   0.000 deg,	R =   90.000 deg
};
P[244]{
   GP1:
	UF : 0, UT : 6,		CONFIG : 'N U T, 0, 0, 0',
	X =  215.585  mm,	Y =   -504.662  mm,	Z =   -269.382  mm,
	W =  90.000 deg,	P =   0.000 deg,	R =   90.000 deg
};
P[245]{
   GP1:
	UF : 0, UT : 6,		CONFIG : 'N U T, 0, 0, 0',
	X =  216.347  mm,	Y =   -504.236  mm,	Z =   -269.297  mm,
	W =  90.000 deg,	P =   0.000 deg,	R =   90.000 deg
};
P[246]{
   GP1:
	UF : 0, UT : 6,		CONFIG : 'N U T, 0, 0, 0',
	X =  218.641  mm,	Y =   -502.952  mm,	Z =   -269.049  mm,
	W =  90.000 deg,	P =   0.000 deg,	R =   90.000 deg
};
P[247]{
   GP1:
	UF : 0, UT : 6,		CONFIG : 'N U T, 0, 0, 0',
	X =  221.310  mm,	Y =   -501.367  mm,	Z =   -269.324  mm,
	W =  90.000 deg,	P =   0.000 deg,	R =   90.000 deg
};
P[248]{
   GP1:
	UF : 0, UT : 6,		CONFIG : 'N U T, 0, 0, 0',
	X =  221.906  mm,	Y =   -501.012  mm,	Z =   -269.387  mm,
	W =  90.000 deg,	P =   0.000 deg,	R =   90.000 deg
};
P[249]{
   GP1:
	UF : 0, UT : 6,		CONFIG : 'N U T, 0, 0, 0',
	X =  222.519  mm,	Y =   -500.699  mm,	Z =   -269.138  mm,
	W =  90.000 deg,	P =   0.000 deg,	R =   90.000 deg
};
P[250]{
   GP1:
	UF : 0, UT : 6,		CONFIG : 'N U T, 0, 0, 0',
	X =  223.411  mm,	Y =   -500.170  mm,	Z =   -269.216  mm,
	W =  90.000 deg,	P =   0.000 deg,	R =   90.000 deg
};
P[251]{
   GP1:
	UF : 0, UT : 6,		CONFIG : 'N U T, 0, 0, 0',
	X =  226.003  mm,	Y =   -498.657  mm,	Z =   -269.323  mm,
	W =  90.000 deg,	P =   0.000 deg,	R =   90.000 deg
};
P[252]{
   GP1:
	UF : 0, UT : 6,		CONFIG : 'N U T, 0, 0, 0',
	X =  228.256  mm,	Y =   -497.360  mm,	Z =   -269.296  mm,
	W =  90.000 deg,	P =   0.000 deg,	R =   90.000 deg
};
P[253]{
   GP1:
	UF : 0, UT : 6,		CONFIG : 'N U T, 0, 0, 0',
	X =  229.072  mm,	Y =   -496.876  mm,	Z =   -269.374  mm,
	W =  90.000 deg,	P =   0.000 deg,	R =   90.000 deg
};
P[254]{
   GP1:
	UF : 0, UT : 6,		CONFIG : 'N U T, 0, 0, 0',
	X =  230.210  mm,	Y =   -496.208  mm,	Z =   -269.446  mm,
	W =  90.000 deg,	P =   0.000 deg,	R =   90.000 deg
};
P[255]{
   GP1:
	UF : 0, UT : 6,		CONFIG : 'N U T, 0, 0, 0',
	X =  230.883  mm,	Y =   -495.859  mm,	Z =   -269.199  mm,
	W =  90.000 deg,	P =   0.000 deg,	R =   90.000 deg
};
P[256]{
   GP1:
	UF : 0, UT : 6,		CONFIG : 'N U T, 0, 0, 0',
	X =  232.254  mm,	Y =   -495.061  mm,	Z =   -269.239  mm,
	W =  90.000 deg,	P =   0.000 deg,	R =   90.000 deg
};
P[257]{
   GP1:
	UF : 0, UT : 6,		CONFIG : 'N U T, 0, 0, 0',
	X =  235.584  mm,	Y =   -493.111  mm,	Z =   -269.410  mm,
	W =  90.000 deg,	P =   0.000 deg,	R =   90.000 deg
};
P[258]{
   GP1:
	UF : 0, UT : 6,		CONFIG : 'N U T, 0, 0, 0',
	X =  236.498  mm,	Y =   -492.647  mm,	Z =   -269.014  mm,
	W =  90.000 deg,	P =   0.000 deg,	R =   90.000 deg
};
P[259]{
   GP1:
	UF : 0, UT : 6,		CONFIG : 'N U T, 0, 0, 0',
	X =  237.109  mm,	Y =   -492.260  mm,	Z =   -269.224  mm,
	W =  90.000 deg,	P =   0.000 deg,	R =   90.000 deg
};
P[260]{
   GP1:
	UF : 0, UT : 6,		CONFIG : 'N U T, 0, 0, 0',
	X =  238.766  mm,	Y =   -491.313  mm,	Z =   -269.165  mm,
	W =  90.000 deg,	P =   0.000 deg,	R =   90.000 deg
};
P[261]{
   GP1:
	UF : 0, UT : 6,		CONFIG : 'N U T, 0, 0, 0',
	X =  240.126  mm,	Y =   -490.546  mm,	Z =   -269.052  mm,
	W =  90.000 deg,	P =   0.000 deg,	R =   90.000 deg
};
P[262]{
   GP1:
	UF : 0, UT : 6,		CONFIG : 'N U T, 0, 0, 0',
	X =  241.507  mm,	Y =   -489.694  mm,	Z =   -269.387  mm,
	W =  90.000 deg,	P =   0.000 deg,	R =   90.000 deg
};
P[263]{
   GP1:
	UF : 0, UT : 6,		CONFIG : 'N U T, 0, 0, 0',
	X =  242.273  mm,	Y =   -489.265  mm,	Z =   -269.307  mm,
	W =  90.000 deg,	P =   0.000 deg,	R =   90.000 deg
};
P[264]{
   GP1:
	UF : 0, UT : 6,		CONFIG : 'N U T, 0, 0, 0',
	X =  243.632  mm,	Y =   -488.480  mm,	Z =   -269.313  mm,
	W =  90.000 deg,	P =   0.000 deg,	R =   90.000 deg
};
P[265]{
   GP1:
	UF : 0, UT : 6,		CONFIG : 'N U T, 0, 0, 0',
	X =  245.660  mm,	Y =   -487.314  mm,	Z =   -269.276  mm,
	W =  90.000 deg,	P =   0.000 deg,	R =   90.000 deg
};
P[266]{
   GP1:
	UF : 0, UT : 6,		CONFIG : 'N U T, 0, 0, 0',
	X =  246.771  mm,	Y =   -486.685  mm,	Z =   -269.204  mm,
	W =  90.000 deg,	P =   0.000 deg,	R =   90.000 deg
};
P[267]{
   GP1:
	UF : 0, UT : 6,		CONFIG : 'N U T, 0, 0, 0',
	X =  248.352  mm,	Y =   -485.803  mm,	Z =   -269.017  mm,
	W =  90.000 deg,	P =   0.000 deg,	R =   90.000 deg
};
P[268]{
   GP1:
	UF : 0, UT : 6,		CONFIG : 'N U T, 0, 0, 0',
	X =  251.132  mm,	Y =   -484.200  mm,	Z =   -269.001  mm,
	W =  90.000 deg,	P =   0.000 deg,	R =   90.000 deg
};
P[269]{
   GP1:
	UF : 0, UT : 6,		CONFIG : 'N U T, 0, 0, 0',
	X =  252.047  mm,	Y =   -483.617  mm,	Z =   -269.338  mm,
	W =  90.000 deg,	P =   0.000 deg,	R =   90.000 deg
};
P[270]{
   GP1:
	UF : 0, UT : 6,		CONFIG : 'N U T, 0, 0, 0',
	X =  253.134  mm,	Y =   -482.971  mm,	Z =   -269.455  mm,
	W =  90.000 deg,	P =   0.000 deg,	R =   90.000 deg
};
P[271]{
   GP1:
	UF : 0, UT : 6,		CONFIG : 'N U T, 0, 0, 0',
	X =  254.223  mm,	Y =   -482.353  mm,	Z =   -269.385  mm,
	W =  90.000 deg,	P =   0.000 deg,	R =   90.000 deg
};
P[272]{
   GP1:
	UF : 0, UT : 6,		CONFIG : 'N U T, 0, 0, 0',
	X =  254.848  mm,	Y =   -482.015  mm,	Z =   -269.242  mm,
	W =  90.000 deg,	P =   0.000 deg,	R =   90.000 deg
};
P[273]{
   GP1:
	UF : 0, UT : 6,		CONFIG : 'N U T, 0, 0, 0',
	X =  255.551  mm,	Y =   -481.595  mm,	Z =   -269.329  mm,
	W =  90.000 deg,	P =   0.000 deg,	R =   90.000 deg
};
P[274]{
   GP1:
	UF : 0, UT : 6,		CONFIG : 'N U T, 0, 0, 0',
	X =  256.403  mm,	Y =   -481.101  mm,	Z =   -269.341  mm,
	W =  90.000 deg,	P =   0.000 deg,	R =   90.000 deg
};
P[275]{
   GP1:
	UF : 0, UT : 6,		CONFIG : 'N U T, 0, 0, 0',
	X =  259.710  mm,	Y =   -479.236  mm,	Z =   -269.065  mm,
	W =  90.000 deg,	P =   0.000 deg,	R =   90.000 deg
};
P[276]{
   GP1:
	UF : 0, UT : 6,		CONFIG : 'N U T, 0, 0, 0',
	X =  260.536  mm,	Y =   -478.706  mm,	Z =   -269.396  mm,
	W =  90.000 deg,	P =   0.000 deg,	R =   90.000 deg
};
P[277]{
   GP1:
	UF : 0, UT : 6,		CONFIG : 'N U T, 0, 0, 0',
	X =  261.985  mm,	Y =   -477.894  mm,	Z =   -269.244  mm,
	W =  90.000 deg,	P =   0.000 deg,	R =   90.000 deg
};
P[278]{
   GP1:
	UF : 0, UT : 6,		CONFIG : 'N U T, 0, 0, 0',
	X =  262.929  mm,	Y =   -477.339  mm,	Z =   -269.304  mm,
	W =  90.000 deg,	P =   0.000 deg,	R =   90.000 deg
};
P[279]{
   GP1:
	UF : 0, UT : 6,		CONFIG : 'N U T, 0, 0, 0',
	X =  264.047  mm,	Y =   -476.690  mm,	Z =   -269.331  mm,
	W =  90.000 deg,	P =   0.000 deg,	R =   90.000 deg
};
P[280]{
   GP1:
	UF : 0, UT : 6,		CONFIG : 'N U T, 0, 0, 0',
	X =  266.437  mm,	Y =   -475.356  mm,	Z =   -269.038  mm,
	W =  90.000 deg,	P =   0.000 deg,	R =   90.000 deg
};
P[281]{
   GP1:
	UF : 0, UT : 6,		CONFIG : 'N U T, 0, 0, 0',
	X =  267.512  mm,	Y =   -474.696  mm,	Z =   -269.291  mm,
	W =  90.000 deg,	P =   0.000 deg,	R =   90.000 deg
};
P[282]{
   GP1:
	UF : 0, UT : 6,		CONFIG : 'N U T, 0, 0, 0',
	X =  269.041  mm,	Y =   -473.840  mm,	Z =   -269.116  mm,
	W =  90.000 deg,	P =   0.000 deg,	R =   90.000 deg
};
P[283]{
   GP1:
	UF : 0, UT : 6,		CONFIG : 'N U T, 0, 0, 0',
	X =  269.847  mm,	Y =   -473.345  mm,	Z =   -269.302  mm,
	W =  90.000 deg,	P =   0.000 deg,	R =   90.000 deg
};
P[284]{
   GP1:
	UF : 0, UT : 6,		CONFIG : 'N U T, 0, 0, 0',
	X =  271.666  mm,	Y =   -472.296  mm,	Z =   -269.293  mm,
	W =  90.000 deg,	P =   0.000 deg,	R =   90.000 deg
};
P[285]{
   GP1:
	UF : 0, UT : 6,		CONFIG : 'N U T, 0, 0, 0',
	X =  272.277  mm,	Y =   -471.925  mm,	Z =   -269.411  mm,
	W =  90.000 deg,	P =   0.000 deg,	R =   90.000 deg
};
P[286]{
   GP1:
	UF : 0, UT : 6,		CONFIG : 'N U T, 0, 0, 0',
	X =  273.298  mm,	Y =   -471.333  mm,	Z =   -269.420  mm,
	W =  90.000 deg,	P =   0.000 deg,	R =   90.000 deg
};
P[287]{
   GP1:
	UF : 0, UT : 6,		CONFIG : 'N U T, 0, 0, 0',
	X =  274.147  mm,	Y =   -470.878  mm,	Z =   -269.207  mm,
	W =  90.000 deg,	P =   0.000 deg,	R =   90.000 deg
};
P[288]{
   GP1:
	UF : 0, UT : 6,		CONFIG : 'N U T, 0, 0, 0',
	X =  274.856  mm,	Y =   -470.428  mm,	Z =   -269.451  mm,
	W =  90.000 deg,	P =   0.000 deg,	R =   90.000 deg
};
P[289]{
   GP1:
	UF : 0, UT : 6,		CONFIG : 'N U T, 0, 0, 0',
	X =  277.033  mm,	Y =   -469.241  mm,	Z =   -269.019  mm,
	W =  90.000 deg,	P =   0.000 deg,	R =   90.000 deg
};
P[290]{
   GP1:
	UF : 0, UT : 6,		CONFIG : 'N U T, 0, 0, 0',
	X =  277.924  mm,	Y =   -468.715  mm,	Z =   -269.099  mm,
	W =  90.000 deg,	P =   0.000 deg,	R =   90.000 deg
};
P[291]{
   GP1:
	UF : 0, UT : 6,		CONFIG : 'N U T, 0, 0, 0',
	X =  280.525  mm,	Y =   -467.156  mm,	Z =   -269.448  mm,
	W =  90.000 deg,	P =   0.000 deg,	R =   90.000 deg
};
P[292]{
   GP1:
	UF : 0, UT : 6,		CONFIG : 'N U T, 0, 0, 0',
	X =  282.234  mm,	Y =   -466.246  mm,	Z =   -268.974  mm,
	W =  90.000 deg,	P =   0.000 deg,	R =   90.000 deg
};
P[293]{
   GP1:
	UF : 0, UT : 6,		CONFIG : 'N U T, 0, 0, 0',
	X =  282.723  mm,	Y =   -465.903  mm,	Z =   -269.346  mm,
	W =  90.000 deg,	P =   0.000 deg,	R =   90.000 deg
};
P[294]{
   GP1:
	UF : 0, UT : 6,		CONFIG : 'N U T, 0, 0, 0',
	X =  283.529  mm,	Y =   -465.432  mm,	Z =   -269.383  mm,
	W =  90.000 deg,	P =   0.000 deg,	R =   90.000 deg
};
P[295]{
   GP1:
	UF : 0, UT : 6,		CONFIG : 'N U T, 0, 0, 0',
	X =  284.424  mm,	Y =   -464.963  mm,	Z =   -269.090  mm,
	W =  90.000 deg,	P =   0.000 deg,	R =   90.000 deg
};
P[296]{
   GP1:
	UF : 0, UT : 6,		CONFIG : 'N U T, 0, 0, 0',
	X =  285.006  mm,	Y =   -464.600  mm,	Z =   -269.256  mm,
	W =  90.000 deg,	P =   0.000 deg,	R =   90.000 deg
};
P[297]{
   GP1:
	UF : 0, UT : 6,		CONFIG : 'N U T, 0, 0, 0',
	X =  286.864  mm,	Y =   -463.526  mm,	Z =   -269.264  mm,
	W =  90.000 deg,	P =   0.000 deg,	R =   90.000 deg
};
P[298]{
   GP1:
	UF : 0, UT : 6,		CONFIG : 'N U T, 0, 0, 0',
	X =  292.273  mm,	Y =   -460.415  mm,	Z =   -269.191  mm,
	W =  90.000 deg,	P =   0.000 deg,	R =   90.000 deg
};
P[299]{
   GP1:
	UF : 0, UT : 6,		CONFIG : 'N U T, 0, 0, 0',
	X =  293.129  mm,	Y =   -459.899  mm,	Z =   -269.320  mm,
	W =  90.000 deg,	P =   0.000 deg,	R =   90.000 deg
};
P[300]{
   GP1:
	UF : 0, UT : 6,		CONFIG : 'N U T, 0, 0, 0',
	X =  295.622  mm,	Y =   -458.443  mm,	Z =   -269.426  mm,
	W =  90.000 deg,	P =   0.000 deg,	R =   90.000 deg
};
P[301]{
   GP1:
	UF : 0, UT : 6,		CONFIG : 'N U T, 0, 0, 0',
	X =  296.281  mm,	Y =   -458.121  mm,	Z =   -269.064  mm,
	W =  90.000 deg,	P =   0.000 deg,	R =   90.000 deg
};
P[302]{
   GP1:
	UF : 0, UT : 6,		CONFIG : 'N U T, 0, 0, 0',
	X =  297.359  mm,	Y =   -457.472  mm,	Z =   -269.232  mm,
	W =  90.000 deg,	P =   0.000 deg,	R =   90.000 deg
};
P[303]{
   GP1:
	UF : 0, UT : 6,		CONFIG : 'N U T, 0, 0, 0',
	X =  298.908  mm,	Y =   -456.564  mm,	Z =   -269.311  mm,
	W =  90.000 deg,	P =   0.000 deg,	R =   90.000 deg
};
P[304]{
   GP1:
	UF : 0, UT : 6,		CONFIG : 'N U T, 0, 0, 0',
	X =  300.417  mm,	Y =   -455.693  mm,	Z =   -269.312  mm,
	W =  90.000 deg,	P =   0.000 deg,	R =   90.000 deg
};
P[305]{
   GP1:
	UF : 0, UT : 6,		CONFIG : 'N U T, 0, 0, 0',
	X =  301.578  mm,	Y =   -455.027  mm,	Z =   -269.285  mm,
	W =  90.000 deg,	P =   0.000 deg,	R =   90.000 deg
};
P[306]{
   GP1:
	UF : 0, UT : 6,		CONFIG : 'N U T, 0, 0, 0',
	X =  302.625  mm,	Y =   -454.401  mm,	Z =   -269.413  mm,
	W =  90.000 deg,	P =   0.000 deg,	R =   90.000 deg
};
P[307]{
   GP1:
	UF : 0, UT : 6,		CONFIG : 'N U T, 0, 0, 0',
	X =  303.606  mm,	Y =   -453.862  mm,	Z =   -269.250  mm,
	W =  90.000 deg,	P =   0.000 deg,	R =   90.000 deg
};
P[308]{
   GP1:
	UF : 0, UT : 6,		CONFIG : 'N U T, 0, 0, 0',
	X =  304.523  mm,	Y =   -453.302  mm,	Z =   -269.437  mm,
	W =  90.000 deg,	P =   0.000 deg,	R =   90.000 deg
};
P[309]{
   GP1:
	UF : 0, UT : 6,		CONFIG : 'N U T, 0, 0, 0',
	X =  305.162  mm,	Y =   -452.948  mm,	Z =   -269.339  mm,
	W =  90.000 deg,	P =   0.000 deg,	R =   90.000 deg
};
P[310]{
   GP1:
	UF : 0, UT : 6,		CONFIG : 'N U T, 0, 0, 0',
	X =  305.828  mm,	Y =   -452.597  mm,	Z =   -269.137  mm,
	W =  90.000 deg,	P =   0.000 deg,	R =   90.000 deg
};
P[311]{
   GP1:
	UF : 0, UT : 6,		CONFIG : 'N U T, 0, 0, 0',
	X =  313.352  mm,	Y =   -448.202  mm,	Z =   -269.449  mm,
	W =  90.000 deg,	P =   0.000 deg,	R =   90.000 deg
};
P[312]{
   GP1:
	UF : 0, UT : 6,		CONFIG : 'N U T, 0, 0, 0',
	X =  315.460  mm,	Y =   -447.035  mm,	Z =   -269.137  mm,
	W =  90.000 deg,	P =   0.000 deg,	R =   90.000 deg
};
P[313]{
   GP1:
	UF : 0, UT : 6,		CONFIG : 'N U T, 0, 0, 0',
	X =  316.338  mm,	Y =   -446.536  mm,	Z =   -269.094  mm,
	W =  90.000 deg,	P =   0.000 deg,	R =   90.000 deg
};
P[314]{
   GP1:
	UF : 0, UT : 6,		CONFIG : 'N U T, 0, 0, 0',
	X =  317.189  mm,	Y =   -446.002  mm,	Z =   -269.358  mm,
	W =  90.000 deg,	P =   0.000 deg,	R =   90.000 deg
};
P[315]{
   GP1:
	UF : 0, UT : 6,		CONFIG : 'N U T, 0, 0, 0',
	X =  318.150  mm,	Y =   -445.433  mm,	Z =   -269.443  mm,
	W =  90.000 deg,	P =   0.000 deg,	R =   90.000 deg
};
P[316]{
   GP1:
	UF : 0, UT : 6,		CONFIG : 'N U T, 0, 0, 0',
	X =  318.811  mm,	Y =   -445.083  mm,	Z =   -269.241  mm,
	W =  90.000 deg,	P =   0.000 deg,	R =   90.000 deg
};
P[317]{
   GP1:
	UF : 0, UT : 6,		CONFIG : 'N U T, 0, 0, 0',
	X =  320.358  mm,	Y =   -444.174  mm,	Z =   -269.341  mm,
	W =  90.000 deg,	P =   0.000 deg,	R =   90.000 deg
};
P[318]{
   GP1:
	UF : 0, UT : 6,		CONFIG : 'N U T, 0, 0, 0',
	X =  321.073  mm,	Y =   -443.751  mm,	Z =   -269.410  mm,
	W =  90.000 deg,	P =   0.000 deg,	R =   90.000 deg
};
P[319]{
   GP1:
	UF : 0, UT : 6,		CONFIG : 'N U T, 0, 0, 0',
	X =  321.804  mm,	Y =   -443.357  mm,	Z =   -269.233  mm,
	W =  90.000 deg,	P =   0.000 deg,	R =   90.000 deg
};
P[320]{
   GP1:
	UF : 0, UT : 6,		CONFIG : 'N U T, 0, 0, 0',
	X =  322.749  mm,	Y =   -442.822  mm,	Z =   -269.163  mm,
	W =  90.000 deg,	P =   0.000 deg,	R =   90.000 deg
};
P[321]{
   GP1:
	UF : 0, UT : 6,		CONFIG : 'N U T, 0, 0, 0',
	X =  323.800  mm,	Y =   -442.187  mm,	Z =   -269.339  mm,
	W =  90.000 deg,	P =   0.000 deg,	R =   90.000 deg
};
P[322]{
   GP1:
	UF : 0, UT : 6,		CONFIG : 'N U T, 0, 0, 0',
	X =  325.285  mm,	Y =   -441.330  mm,	Z =   -269.336  mm,
	W =  90.000 deg,	P =   0.000 deg,	R =   90.000 deg
};
P[323]{
   GP1:
	UF : 0, UT : 6,		CONFIG : 'N U T, 0, 0, 0',
	X =  326.078  mm,	Y =   -440.863  mm,	Z =   -269.393  mm,
	W =  90.000 deg,	P =   0.000 deg,	R =   90.000 deg
};
P[324]{
   GP1:
	UF : 0, UT : 6,		CONFIG : 'N U T, 0, 0, 0',
	X =  326.982  mm,	Y =   -440.357  mm,	Z =   -269.296  mm,
	W =  90.000 deg,	P =   0.000 deg,	R =   90.000 deg
};
P[325]{
   GP1:
	UF : 0, UT : 6,		CONFIG : 'N U T, 0, 0, 0',
	X =  327.755  mm,	Y =   -439.936  mm,	Z =   -269.142  mm,
	W =  90.000 deg,	P =   0.000 deg,	R =   90.000 deg
};
P[326]{
   GP1:
	UF : 0, UT : 6,		CONFIG : 'N U T, 0, 0, 0',
	X =  329.364  mm,	Y =   -439.014  mm,	Z =   -269.099  mm,
	W =  90.000 deg,	P =   0.000 deg,	R =   90.000 deg
};
P[327]{
   GP1:
	UF : 0, UT : 6,		CONFIG : 'N U T, 0, 0, 0',
	X =  330.108  mm,	Y =   -438.558  mm,	Z =   -269.256  mm,
	W =  90.000 deg,	P =   0.000 deg,	R =   90.000 deg
};
P[328]{
   GP1:
	UF : 0, UT : 6,		CONFIG : 'N U T, 0, 0, 0',
	X =  331.540  mm,	Y =   -437.727  mm,	Z =   -269.286  mm,
	W =  90.000 deg,	P =   0.000 deg,	R =   90.000 deg
};
P[329]{
   GP1:
	UF : 0, UT : 6,		CONFIG : 'N U T, 0, 0, 0',
	X =  332.442  mm,	Y =   -437.196  mm,	Z =   -269.346  mm,
	W =  90.000 deg,	P =   0.000 deg,	R =   90.000 deg
};
P[330]{
   GP1:
	UF : 0, UT : 6,		CONFIG : 'N U T, 0, 0, 0',
	X =  334.336  mm,	Y =   -436.163  mm,	Z =   -268.973  mm,
	W =  90.000 deg,	P =   0.000 deg,	R =   90.000 deg
};
P[331]{
   GP1:
	UF : 0, UT : 6,		CONFIG : 'N U T, 0, 0, 0',
	X =  335.413  mm,	Y =   -435.525  mm,	Z =   -269.070  mm,
	W =  90.000 deg,	P =   0.000 deg,	R =   90.000 deg
};
P[332]{
   GP1:
	UF : 0, UT : 6,		CONFIG : 'N U T, 0, 0, 0',
	X =  336.278  mm,	Y =   -434.994  mm,	Z =   -269.267  mm,
	W =  90.000 deg,	P =   0.000 deg,	R =   90.000 deg
};
P[333]{
   GP1:
	UF : 0, UT : 6,		CONFIG : 'N U T, 0, 0, 0',
	X =  339.387  mm,	Y =   -433.175  mm,	Z =   -269.413  mm,
	W =  90.000 deg,	P =   0.000 deg,	R =   90.000 deg
};
P[334]{
   GP1:
	UF : 0, UT : 6,		CONFIG : 'N U T, 0, 0, 0',
	X =  340.335  mm,	Y =   -432.626  mm,	Z =   -269.428  mm,
	W =  90.000 deg,	P =   0.000 deg,	R =   90.000 deg
};
P[335]{
   GP1:
	UF : 0, UT : 6,		CONFIG : 'N U T, 0, 0, 0',
	X =  341.311  mm,	Y =   -432.061  mm,	Z =   -269.433  mm,
	W =  90.000 deg,	P =   0.000 deg,	R =   90.000 deg
};
P[336]{
   GP1:
	UF : 0, UT : 6,		CONFIG : 'N U T, 0, 0, 0',
	X =  342.106  mm,	Y =   -431.604  mm,	Z =   -269.424  mm,
	W =  90.000 deg,	P =   0.000 deg,	R =   90.000 deg
};
P[337]{
   GP1:
	UF : 0, UT : 6,		CONFIG : 'N U T, 0, 0, 0',
	X =  342.943  mm,	Y =   -431.138  mm,	Z =   -269.319  mm,
	W =  90.000 deg,	P =   0.000 deg,	R =   90.000 deg
};
P[338]{
   GP1:
	UF : 0, UT : 6,		CONFIG : 'N U T, 0, 0, 0',
	X =  343.749  mm,	Y =   -430.653  mm,	Z =   -269.435  mm,
	W =  90.000 deg,	P =   0.000 deg,	R =   90.000 deg
};
P[339]{
   GP1:
	UF : 0, UT : 6,		CONFIG : 'N U T, 0, 0, 0',
	X =  344.298  mm,	Y =   -430.405  mm,	Z =   -269.016  mm,
	W =  90.000 deg,	P =   0.000 deg,	R =   90.000 deg
};
P[340]{
   GP1:
	UF : 0, UT : 6,		CONFIG : 'N U T, 0, 0, 0',
	X =  345.145  mm,	Y =   -429.864  mm,	Z =   -269.335  mm,
	W =  90.000 deg,	P =   0.000 deg,	R =   90.000 deg
};
P[341]{
   GP1:
	UF : 0, UT : 6,		CONFIG : 'N U T, 0, 0, 0',
	X =  346.056  mm,	Y =   -429.330  mm,	Z =   -269.380  mm,
	W =  90.000 deg,	P =   0.000 deg,	R =   90.000 deg
};
P[342]{
   GP1:
	UF : 0, UT : 6,		CONFIG : 'N U T, 0, 0, 0',
	X =  347.425  mm,	Y =   -428.590  mm,	Z =   -269.065  mm,
	W =  90.000 deg,	P =   0.000 deg,	R =   90.000 deg
};
P[343]{
   GP1:
	UF : 0, UT : 6,		CONFIG : 'N U T, 0, 0, 0',
	X =  348.256  mm,	Y =   -428.091  mm,	Z =   -269.184  mm,
	W =  90.000 deg,	P =   0.000 deg,	R =   90.000 deg
};
P[344]{
   GP1:
	UF : 0, UT : 6,		CONFIG : 'N U T, 0, 0, 0',
	X =  349.062  mm,	Y =   -427.606  mm,	Z =   -269.309  mm,
	W =  90.000 deg,	P =   0.000 deg,	R =   90.000 deg
};
P[345]{
   GP1:
	UF : 0, UT : 6,		CONFIG : 'N U T, 0, 0, 0',
	X =  350.004  mm,	Y =   -427.059  mm,	Z =   -269.329  mm,
	W =  90.000 deg,	P =   0.000 deg,	R =   90.000 deg
};
P[346]{
   GP1:
	UF : 0, UT : 6,		CONFIG : 'N U T, 0, 0, 0',
	X =  352.372  mm,	Y =   -425.692  mm,	Z =   -269.327  mm,
	W =  90.000 deg,	P =   0.000 deg,	R =   90.000 deg
};
P[347]{
   GP1:
	UF : 0, UT : 6,		CONFIG : 'N U T, 0, 0, 0',
	X =  354.004  mm,	Y =   -424.776  mm,	Z =   -269.167  mm,
	W =  90.000 deg,	P =   0.000 deg,	R =   90.000 deg
};
P[348]{
   GP1:
	UF : 0, UT : 6,		CONFIG : 'N U T, 0, 0, 0',
	X =  355.765  mm,	Y =   -423.737  mm,	Z =   -269.305  mm,
	W =  90.000 deg,	P =   0.000 deg,	R =   90.000 deg
};
P[349]{
   GP1:
	UF : 0, UT : 6,		CONFIG : 'N U T, 0, 0, 0',
	X =  357.421  mm,	Y =   -422.832  mm,	Z =   -268.988  mm,
	W =  90.000 deg,	P =   0.000 deg,	R =   90.000 deg
};
P[350]{
   GP1:
	UF : 0, UT : 6,		CONFIG : 'N U T, 0, 0, 0',
	X =  358.031  mm,	Y =   -422.421  mm,	Z =   -269.347  mm,
	W =  90.000 deg,	P =   0.000 deg,	R =   90.000 deg
};
P[351]{
   GP1:
	UF : 0, UT : 6,		CONFIG : 'N U T, 0, 0, 0',
	X =  358.650  mm,	Y =   -422.122  mm,	Z =   -268.987  mm,
	W =  90.000 deg,	P =   0.000 deg,	R =   90.000 deg
};
P[352]{
   GP1:
	UF : 0, UT : 6,		CONFIG : 'N U T, 0, 0, 0',
	X =  359.498  mm,	Y =   -421.575  mm,	Z =   -269.342  mm,
	W =  90.000 deg,	P =   0.000 deg,	R =   90.000 deg
};
P[353]{
   GP1:
	UF : 0, UT : 6,		CONFIG : 'N U T, 0, 0, 0',
	X =  360.390  mm,	Y =   -421.079  mm,	Z =   -269.221  mm,
	W =  90.000 deg,	P =   0.000 deg,	R =   90.000 deg
};
P[354]{
   GP1:
	UF : 0, UT : 6,		CONFIG : 'N U T, 0, 0, 0',
	X =  361.200  mm,	Y =   -420.629  mm,	Z =   -269.112  mm,
	W =  90.000 deg,	P =   0.000 deg,	R =   90.000 deg
};
P[355]{
   GP1:
	UF : 0, UT : 6,		CONFIG : 'N U T, 0, 0, 0',
	X =  361.891  mm,	Y =   -420.226  mm,	Z =   -269.136  mm,
	W =  90.000 deg,	P =   0.000 deg,	R =   90.000 deg
};
P[356]{
   GP1:
	UF : 0, UT : 6,		CONFIG : 'N U T, 0, 0, 0',
	X =  363.624  mm,	Y =   -419.196  mm,	Z =   -269.324  mm,
	W =  90.000 deg,	P =   0.000 deg,	R =   90.000 deg
};
P[357]{
   GP1:
	UF : 0, UT : 6,		CONFIG : 'N U T, 0, 0, 0',
	X =  364.398  mm,	Y =   -418.610  mm,	Z =   -269.317  mm,
	W =  90.000 deg,	P =   0.000 deg,	R =   90.000 deg
};
P[358]{
   GP1:
	UF : 0, UT : 6,		CONFIG : 'N U T, 0, 0, 0',
	X =  365.526  mm,	Y =   -416.752  mm,	Z =   -269.406  mm,
	W =  90.000 deg,	P =   0.000 deg,	R =   90.000 deg
};
P[359]{
   GP1:
	UF : 0, UT : 6,		CONFIG : 'N U T, 0, 0, 0',
	X =  365.595  mm,	Y =   -414.726  mm,	Z =   -269.333  mm,
	W =  90.000 deg,	P =   0.000 deg,	R =   90.000 deg
};
P[360]{
   GP1:
	UF : 0, UT : 6,		CONFIG : 'N U T, 0, 0, 0',
	X =  365.145  mm,	Y =   -413.589  mm,	Z =   -269.367  mm,
	W =  90.000 deg,	P =   0.000 deg,	R =   90.000 deg
};
P[361]{
   GP1:
	UF : 0, UT : 6,		CONFIG : 'N U T, 0, 0, 0',
	X =  364.689  mm,	Y =   -412.774  mm,	Z =   -269.437  mm,
	W =  90.000 deg,	P =   0.000 deg,	R =   90.000 deg
};
P[362]{
   GP1:
	UF : 0, UT : 6,		CONFIG : 'N U T, 0, 0, 0',
	X =  364.271  mm,	Y =   -411.936  mm,	Z =   -269.025  mm,
	W =  90.000 deg,	P =   0.000 deg,	R =   90.000 deg
};
P[363]{
   GP1:
	UF : 0, UT : 6,		CONFIG : 'N U T, 0, 0, 0',
	X =  363.755  mm,	Y =   -411.123  mm,	Z =   -269.321  mm,
	W =  90.000 deg,	P =   0.000 deg,	R =   90.000 deg
};
P[364]{
   GP1:
	UF : 0, UT : 6,		CONFIG : 'N U T, 0, 0, 0',
	X =  363.197  mm,	Y =   -410.159  mm,	Z =   -269.332  mm,
	W =  90.000 deg,	P =   0.000 deg,	R =   90.000 deg
};
P[365]{
   GP1:
	UF : 0, UT : 6,		CONFIG : 'N U T, 0, 0, 0',
	X =  362.819  mm,	Y =   -409.421  mm,	Z =   -269.028  mm,
	W =  90.000 deg,	P =   0.000 deg,	R =   90.000 deg
};
P[366]{
   GP1:
	UF : 0, UT : 6,		CONFIG : 'N U T, 0, 0, 0',
	X =  361.465  mm,	Y =   -407.171  mm,	Z =   -269.368  mm,
	W =  90.000 deg,	P =   0.000 deg,	R =   90.000 deg
};
P[367]{
   GP1:
	UF : 0, UT : 6,		CONFIG : 'N U T, 0, 0, 0',
	X =  359.085  mm,	Y =   -403.065  mm,	Z =   -269.420  mm,
	W =  90.000 deg,	P =   0.000 deg,	R =   90.000 deg
};
P[368]{
   GP1:
	UF : 0, UT : 6,		CONFIG : 'N U T, 0, 0, 0',
	X =  358.187  mm,	Y =   -401.468  mm,	Z =   -269.275  mm,
	W =  90.000 deg,	P =   0.000 deg,	R =   90.000 deg
};
P[369]{
   GP1:
	UF : 0, UT : 6,		CONFIG : 'N U T, 0, 0, 0',
	X =  355.420  mm,	Y =   -396.726  mm,	Z =   -269.453  mm,
	W =  90.000 deg,	P =   0.000 deg,	R =   90.000 deg
};
P[370]{
   GP1:
	UF : 0, UT : 6,		CONFIG : 'N U T, 0, 0, 0',
	X =  354.962  mm,	Y =   -395.844  mm,	Z =   -269.140  mm,
	W =  90.000 deg,	P =   0.000 deg,	R =   90.000 deg
};
P[371]{
   GP1:
	UF : 0, UT : 6,		CONFIG : 'N U T, 0, 0, 0',
	X =  354.478  mm,	Y =   -395.067  mm,	Z =   -269.356  mm,
	W =  90.000 deg,	P =   0.000 deg,	R =   90.000 deg
};
P[372]{
   GP1:
	UF : 0, UT : 6,		CONFIG : 'N U T, 0, 0, 0',
	X =  353.811  mm,	Y =   -393.850  mm,	Z =   -269.141  mm,
	W =  90.000 deg,	P =   0.000 deg,	R =   90.000 deg
};
P[373]{
   GP1:
	UF : 0, UT : 6,		CONFIG : 'N U T, 0, 0, 0',
	X =  353.179  mm,	Y =   -392.790  mm,	Z =   -269.256  mm,
	W =  90.000 deg,	P =   0.000 deg,	R =   90.000 deg
};
P[374]{
   GP1:
	UF : 0, UT : 6,		CONFIG : 'N U T, 0, 0, 0',
	X =  352.085  mm,	Y =   -390.854  mm,	Z =   -269.114  mm,
	W =  90.000 deg,	P =   0.000 deg,	R =   90.000 deg
};
P[375]{
   GP1:
	UF : 0, UT : 6,		CONFIG : 'N U T, 0, 0, 0',
	X =  351.318  mm,	Y =   -389.576  mm,	Z =   -269.289  mm,
	W =  90.000 deg,	P =   0.000 deg,	R =   90.000 deg
};
P[376]{
   GP1:
	UF : 0, UT : 6,		CONFIG : 'N U T, 0, 0, 0',
	X =  350.382  mm,	Y =   -387.971  mm,	Z =   -269.345  mm,
	W =  90.000 deg,	P =   0.000 deg,	R =   90.000 deg
};
P[377]{
   GP1:
	UF : 0, UT : 6,		CONFIG : 'N U T, 0, 0, 0',
	X =  349.845  mm,	Y =   -386.962  mm,	Z =   -269.066  mm,
	W =  90.000 deg,	P =   0.000 deg,	R =   90.000 deg
};
P[378]{
   GP1:
	UF : 0, UT : 6,		CONFIG : 'N U T, 0, 0, 0',
	X =  348.402  mm,	Y =   -384.536  mm,	Z =   -269.329  mm,
	W =  90.000 deg,	P =   0.000 deg,	R =   90.000 deg
};
P[379]{
   GP1:
	UF : 0, UT : 6,		CONFIG : 'N U T, 0, 0, 0',
	X =  348.092  mm,	Y =   -383.930  mm,	Z =   -269.087  mm,
	W =  90.000 deg,	P =   0.000 deg,	R =   90.000 deg
};
P[380]{
   GP1:
	UF : 0, UT : 6,		CONFIG : 'N U T, 0, 0, 0',
	X =  347.261  mm,	Y =   -382.567  mm,	Z =   -269.358  mm,
	W =  90.000 deg,	P =   0.000 deg,	R =   90.000 deg
};
P[381]{
   GP1:
	UF : 0, UT : 6,		CONFIG : 'N U T, 0, 0, 0',
	X =  346.197  mm,	Y =   -380.688  mm,	Z =   -269.225  mm,
	W =  90.000 deg,	P =   0.000 deg,	R =   90.000 deg
};
P[382]{
   GP1:
	UF : 0, UT : 6,		CONFIG : 'N U T, 0, 0, 0',
	X =  345.280  mm,	Y =   -379.145  mm,	Z =   -269.391  mm,
	W =  90.000 deg,	P =   0.000 deg,	R =   90.000 deg
};
P[383]{
   GP1:
	UF : 0, UT : 6,		CONFIG : 'N U T, 0, 0, 0',
	X =  344.658  mm,	Y =   -378.053  mm,	Z =   -269.339  mm,
	W =  90.000 deg,	P =   0.000 deg,	R =   90.000 deg
};
P[384]{
   GP1:
	UF : 0, UT : 6,		CONFIG : 'N U T, 0, 0, 0',
	X =  344.158  mm,	Y =   -377.149  mm,	Z =   -269.198  mm,
	W =  90.000 deg,	P =   0.000 deg,	R =   90.000 deg
};
P[385]{
   GP1:
	UF : 0, UT : 6,		CONFIG : 'N U T, 0, 0, 0',
	X =  343.702  mm,	Y =   -376.316  mm,	Z =   -269.046  mm,
	W =  90.000 deg,	P =   0.000 deg,	R =   90.000 deg
};
P[386]{
   GP1:
	UF : 0, UT : 6,		CONFIG : 'N U T, 0, 0, 0',
	X =  342.986  mm,	Y =   -375.101  mm,	Z =   -269.135  mm,
	W =  90.000 deg,	P =   0.000 deg,	R =   90.000 deg
};
P[387]{
   GP1:
	UF : 0, UT : 6,		CONFIG : 'N U T, 0, 0, 0',
	X =  342.128  mm,	Y =   -373.653  mm,	Z =   -269.266  mm,
	W =  90.000 deg,	P =   0.000 deg,	R =   90.000 deg
};
P[388]{
   GP1:
	UF : 0, UT : 6,		CONFIG : 'N U T, 0, 0, 0',
	X =  341.473  mm,	Y =   -372.543  mm,	Z =   -269.354  mm,
	W =  90.000 deg,	P =   0.000 deg,	R =   90.000 deg
};
P[389]{
   GP1:
	UF : 0, UT : 6,		CONFIG : 'N U T, 0, 0, 0',
	X =  340.834  mm,	Y =   -371.385  mm,	Z =   -269.172  mm,
	W =  90.000 deg,	P =   0.000 deg,	R =   90.000 deg
};
P[390]{
   GP1:
	UF : 0, UT : 6,		CONFIG : 'N U T, 0, 0, 0',
	X =  340.258  mm,	Y =   -370.430  mm,	Z =   -269.322  mm,
	W =  90.000 deg,	P =   0.000 deg,	R =   90.000 deg
};
P[391]{
   GP1:
	UF : 0, UT : 6,		CONFIG : 'N U T, 0, 0, 0',
	X =  339.718  mm,	Y =   -369.516  mm,	Z =   -269.403  mm,
	W =  90.000 deg,	P =   0.000 deg,	R =   90.000 deg
};
P[392]{
   GP1:
	UF : 0, UT : 6,		CONFIG : 'N U T, 0, 0, 0',
	X =  338.350  mm,	Y =   -367.140  mm,	Z =   -269.376  mm,
	W =  90.000 deg,	P =   0.000 deg,	R =   90.000 deg
};
P[393]{
   GP1:
	UF : 0, UT : 6,		CONFIG : 'N U T, 0, 0, 0',
	X =  337.340  mm,	Y =   -365.380  mm,	Z =   -269.336  mm,
	W =  90.000 deg,	P =   0.000 deg,	R =   90.000 deg
};
P[394]{
   GP1:
	UF : 0, UT : 6,		CONFIG : 'N U T, 0, 0, 0',
	X =  336.168  mm,	Y =   -363.330  mm,	Z =   -269.263  mm,
	W =  90.000 deg,	P =   0.000 deg,	R =   90.000 deg
};
P[395]{
   GP1:
	UF : 0, UT : 6,		CONFIG : 'N U T, 0, 0, 0',
	X =  335.544  mm,	Y =   -362.261  mm,	Z =   -269.304  mm,
	W =  90.000 deg,	P =   0.000 deg,	R =   90.000 deg
};
P[396]{
   GP1:
	UF : 0, UT : 6,		CONFIG : 'N U T, 0, 0, 0',
	X =  334.648  mm,	Y =   -360.644  mm,	Z =   -269.074  mm,
	W =  90.000 deg,	P =   0.000 deg,	R =   90.000 deg
};
P[397]{
   GP1:
	UF : 0, UT : 6,		CONFIG : 'N U T, 0, 0, 0',
	X =  334.085  mm,	Y =   -359.762  mm,	Z =   -269.408  mm,
	W =  90.000 deg,	P =   0.000 deg,	R =   90.000 deg
};
P[398]{
   GP1:
	UF : 0, UT : 6,		CONFIG : 'N U T, 0, 0, 0',
	X =  333.758  mm,	Y =   -359.172  mm,	Z =   -269.323  mm,
	W =  90.000 deg,	P =   0.000 deg,	R =   90.000 deg
};
P[399]{
   GP1:
	UF : 0, UT : 6,		CONFIG : 'N U T, 0, 0, 0',
	X =  333.363  mm,	Y =   -358.478  mm,	Z =   -269.284  mm,
	W =  90.000 deg,	P =   0.000 deg,	R =   90.000 deg
};
P[400]{
   GP1:
	UF : 0, UT : 6,		CONFIG : 'N U T, 0, 0, 0',
	X =  332.306  mm,	Y =   -356.678  mm,	Z =   -269.399  mm,
	W =  90.000 deg,	P =   0.000 deg,	R =   90.000 deg
};
P[401]{
   GP1:
	UF : 0, UT : 6,		CONFIG : 'N U T, 0, 0, 0',
	X =  331.093  mm,	Y =   -354.500  mm,	Z =   -269.124  mm,
	W =  90.000 deg,	P =   0.000 deg,	R =   90.000 deg
};
P[402]{
   GP1:
	UF : 0, UT : 6,		CONFIG : 'N U T, 0, 0, 0',
	X =  330.111  mm,	Y =   -352.836  mm,	Z =   -269.253  mm,
	W =  90.000 deg,	P =   0.000 deg,	R =   90.000 deg
};
P[403]{
   GP1:
	UF : 0, UT : 6,		CONFIG : 'N U T, 0, 0, 0',
	X =  329.654  mm,	Y =   -351.994  mm,	Z =   -269.072  mm,
	W =  90.000 deg,	P =   0.000 deg,	R =   90.000 deg
};
P[404]{
   GP1:
	UF : 0, UT : 6,		CONFIG : 'N U T, 0, 0, 0',
	X =  327.200  mm,	Y =   -347.835  mm,	Z =   -269.396  mm,
	W =  90.000 deg,	P =   0.000 deg,	R =   90.000 deg
};
P[405]{
   GP1:
	UF : 0, UT : 6,		CONFIG : 'N U T, 0, 0, 0',
	X =  326.715  mm,	Y =   -346.938  mm,	Z =   -269.189  mm,
	W =  90.000 deg,	P =   0.000 deg,	R =   90.000 deg
};
P[406]{
   GP1:
	UF : 0, UT : 6,		CONFIG : 'N U T, 0, 0, 0',
	X =  325.883  mm,	Y =   -345.524  mm,	Z =   -269.290  mm,
	W =  90.000 deg,	P =   0.000 deg,	R =   90.000 deg
};
P[407]{
   GP1:
	UF : 0, UT : 6,		CONFIG : 'N U T, 0, 0, 0',
	X =  324.810  mm,	Y =   -343.654  mm,	Z =   -269.253  mm,
	W =  90.000 deg,	P =   0.000 deg,	R =   90.000 deg
};
P[408]{
   GP1:
	UF : 0, UT : 6,		CONFIG : 'N U T, 0, 0, 0',
	X =  323.261  mm,	Y =   -340.975  mm,	Z =   -269.262  mm,
	W =  90.000 deg,	P =   0.000 deg,	R =   90.000 deg
};
P[409]{
   GP1:
	UF : 0, UT : 6,		CONFIG : 'N U T, 0, 0, 0',
	X =  321.362  mm,	Y =   -337.735  mm,	Z =   -269.437  mm,
	W =  90.000 deg,	P =   0.000 deg,	R =   90.000 deg
};
P[410]{
   GP1:
	UF : 0, UT : 6,		CONFIG : 'N U T, 0, 0, 0',
	X =  319.900  mm,	Y =   -335.124  mm,	Z =   -269.157  mm,
	W =  90.000 deg,	P =   0.000 deg,	R =   90.000 deg
};
P[411]{
   GP1:
	UF : 0, UT : 6,		CONFIG : 'N U T, 0, 0, 0',
	X =  318.474  mm,	Y =   -332.714  mm,	Z =   -269.370  mm,
	W =  90.000 deg,	P =   0.000 deg,	R =   90.000 deg
};
P[412]{
   GP1:
	UF : 0, UT : 6,		CONFIG : 'N U T, 0, 0, 0',
	X =  317.045  mm,	Y =   -330.239  mm,	Z =   -269.369  mm,
	W =  90.000 deg,	P =   0.000 deg,	R =   90.000 deg
};
P[413]{
   GP1:
	UF : 0, UT : 6,		CONFIG : 'N U T, 0, 0, 0',
	X =  316.602  mm,	Y =   -329.470  mm,	Z =   -269.367  mm,
	W =  90.000 deg,	P =   0.000 deg,	R =   90.000 deg
};
P[414]{
   GP1:
	UF : 0, UT : 6,		CONFIG : 'N U T, 0, 0, 0',
	X =  316.214  mm,	Y =   -328.794  mm,	Z =   -269.350  mm,
	W =  90.000 deg,	P =   0.000 deg,	R =   90.000 deg
};
P[415]{
   GP1:
	UF : 0, UT : 6,		CONFIG : 'N U T, 0, 0, 0',
	X =  315.838  mm,	Y =   -328.104  mm,	Z =   -269.211  mm,
	W =  90.000 deg,	P =   0.000 deg,	R =   90.000 deg
};
P[416]{
   GP1:
	UF : 0, UT : 6,		CONFIG : 'N U T, 0, 0, 0',
	X =  315.291  mm,	Y =   -327.162  mm,	Z =   -269.228  mm,
	W =  90.000 deg,	P =   0.000 deg,	R =   90.000 deg
};
P[417]{
   GP1:
	UF : 0, UT : 6,		CONFIG : 'N U T, 0, 0, 0',
	X =  314.714  mm,	Y =   -326.100  mm,	Z =   -269.007  mm,
	W =  90.000 deg,	P =   0.000 deg,	R =   90.000 deg
};
P[418]{
   GP1:
	UF : 0, UT : 6,		CONFIG : 'N U T, 0, 0, 0',
	X =  313.999  mm,	Y =   -324.885  mm,	Z =   -269.091  mm,
	W =  90.000 deg,	P =   0.000 deg,	R =   90.000 deg
};
P[419]{
   GP1:
	UF : 0, UT : 6,		CONFIG : 'N U T, 0, 0, 0',
	X =  313.609  mm,	Y =   -324.220  mm,	Z =   -269.123  mm,
	W =  90.000 deg,	P =   0.000 deg,	R =   90.000 deg
};
P[420]{
   GP1:
	UF : 0, UT : 6,		CONFIG : 'N U T, 0, 0, 0',
	X =  312.921  mm,	Y =   -323.069  mm,	Z =   -269.272  mm,
	W =  90.000 deg,	P =   0.000 deg,	R =   90.000 deg
};
P[421]{
   GP1:
	UF : 0, UT : 6,		CONFIG : 'N U T, 0, 0, 0',
	X =  312.100  mm,	Y =   -321.688  mm,	Z =   -269.413  mm,
	W =  90.000 deg,	P =   0.000 deg,	R =   90.000 deg
};
P[422]{
   GP1:
	UF : 0, UT : 6,		CONFIG : 'N U T, 0, 0, 0',
	X =  310.722  mm,	Y =   -319.286  mm,	Z =   -269.365  mm,
	W =  90.000 deg,	P =   0.000 deg,	R =   90.000 deg
};
P[423]{
   GP1:
	UF : 0, UT : 6,		CONFIG : 'N U T, 0, 0, 0',
	X =  310.166  mm,	Y =   -318.334  mm,	Z =   -269.402  mm,
	W =  90.000 deg,	P =   0.000 deg,	R =   90.000 deg
};
P[424]{
   GP1:
	UF : 0, UT : 6,		CONFIG : 'N U T, 0, 0, 0',
	X =  309.650  mm,	Y =   -317.449  mm,	Z =   -269.433  mm,
	W =  90.000 deg,	P =   0.000 deg,	R =   90.000 deg
};
P[425]{
   GP1:
	UF : 0, UT : 6,		CONFIG : 'N U T, 0, 0, 0',
	X =  308.314  mm,	Y =   -315.045  mm,	Z =   -269.110  mm,
	W =  90.000 deg,	P =   0.000 deg,	R =   90.000 deg
};
P[426]{
   GP1:
	UF : 0, UT : 6,		CONFIG : 'N U T, 0, 0, 0',
	X =  307.757  mm,	Y =   -314.075  mm,	Z =   -269.090  mm,
	W =  90.000 deg,	P =   0.000 deg,	R =   90.000 deg
};
P[427]{
   GP1:
	UF : 0, UT : 6,		CONFIG : 'N U T, 0, 0, 0',
	X =  307.235  mm,	Y =   -313.179  mm,	Z =   -269.119  mm,
	W =  90.000 deg,	P =   0.000 deg,	R =   90.000 deg
};
P[428]{
   GP1:
	UF : 0, UT : 6,		CONFIG : 'N U T, 0, 0, 0',
	X =  306.388  mm,	Y =   -311.778  mm,	Z =   -269.357  mm,
	W =  90.000 deg,	P =   0.000 deg,	R =   90.000 deg
};
P[429]{
   GP1:
	UF : 0, UT : 6,		CONFIG : 'N U T, 0, 0, 0',
	X =  305.700  mm,	Y =   -310.564  mm,	Z =   -269.275  mm,
	W =  90.000 deg,	P =   0.000 deg,	R =   90.000 deg
};
P[430]{
   GP1:
	UF : 0, UT : 6,		CONFIG : 'N U T, 0, 0, 0',
	X =  304.561  mm,	Y =   -308.623  mm,	Z =   -269.388  mm,
	W =  90.000 deg,	P =   0.000 deg,	R =   90.000 deg
};
P[431]{
   GP1:
	UF : 0, UT : 6,		CONFIG : 'N U T, 0, 0, 0',
	X =  303.750  mm,	Y =   -307.166  mm,	Z =   -269.196  mm,
	W =  90.000 deg,	P =   0.000 deg,	R =   90.000 deg
};
P[432]{
   GP1:
	UF : 0, UT : 6,		CONFIG : 'N U T, 0, 0, 0',
	X =  301.889  mm,	Y =   -303.975  mm,	Z =   -269.315  mm,
	W =  90.000 deg,	P =   0.000 deg,	R =   90.000 deg
};
P[433]{
   GP1:
	UF : 0, UT : 6,		CONFIG : 'N U T, 0, 0, 0',
	X =  300.610  mm,	Y =   -301.749  mm,	Z =   -269.275  mm,
	W =  90.000 deg,	P =   0.000 deg,	R =   90.000 deg
};
P[434]{
   GP1:
	UF : 0, UT : 6,		CONFIG : 'N U T, 0, 0, 0',
	X =  299.950  mm,	Y =   -300.630  mm,	Z =   -269.364  mm,
	W =  90.000 deg,	P =   0.000 deg,	R =   90.000 deg
};
P[435]{
   GP1:
	UF : 0, UT : 6,		CONFIG : 'N U T, 0, 0, 0',
	X =  299.572  mm,	Y =   -299.940  mm,	Z =   -269.236  mm,
	W =  90.000 deg,	P =   0.000 deg,	R =   90.000 deg
};
P[436]{
   GP1:
	UF : 0, UT : 6,		CONFIG : 'N U T, 0, 0, 0',
	X =  297.512  mm,	Y =   -296.376  mm,	Z =   -269.247  mm,
	W =  90.000 deg,	P =   0.000 deg,	R =   90.000 deg
};
P[437]{
   GP1:
	UF : 0, UT : 6,		CONFIG : 'N U T, 0, 0, 0',
	X =  296.402  mm,	Y =   -294.450  mm,	Z =   -269.234  mm,
	W =  90.000 deg,	P =   0.000 deg,	R =   90.000 deg
};
P[438]{
   GP1:
	UF : 0, UT : 6,		CONFIG : 'N U T, 0, 0, 0',
	X =  296.044  mm,	Y =   -293.837  mm,	Z =   -269.267  mm,
	W =  90.000 deg,	P =   0.000 deg,	R =   90.000 deg
};
P[439]{
   GP1:
	UF : 0, UT : 6,		CONFIG : 'N U T, 0, 0, 0',
	X =  295.568  mm,	Y =   -293.012  mm,	Z =   -269.261  mm,
	W =  90.000 deg,	P =   0.000 deg,	R =   90.000 deg
};
P[440]{
   GP1:
	UF : 0, UT : 6,		CONFIG : 'N U T, 0, 0, 0',
	X =  292.809  mm,	Y =   -288.214  mm,	Z =   -269.195  mm,
	W =  90.000 deg,	P =   0.000 deg,	R =   90.000 deg
};
P[441]{
   GP1:
	UF : 0, UT : 6,		CONFIG : 'N U T, 0, 0, 0',
	X =  292.169  mm,	Y =   -287.105  mm,	Z =   -269.193  mm,
	W =  90.000 deg,	P =   0.000 deg,	R =   90.000 deg
};
P[442]{
   GP1:
	UF : 0, UT : 6,		CONFIG : 'N U T, 0, 0, 0',
	X =  291.600  mm,	Y =   -286.160  mm,	Z =   -269.327  mm,
	W =  90.000 deg,	P =   0.000 deg,	R =   90.000 deg
};
P[443]{
   GP1:
	UF : 0, UT : 6,		CONFIG : 'N U T, 0, 0, 0',
	X =  291.204  mm,	Y =   -285.432  mm,	Z =   -269.184  mm,
	W =  90.000 deg,	P =   0.000 deg,	R =   90.000 deg
};
P[444]{
   GP1:
	UF : 0, UT : 6,		CONFIG : 'N U T, 0, 0, 0',
	X =  290.764  mm,	Y =   -284.705  mm,	Z =   -269.305  mm,
	W =  90.000 deg,	P =   0.000 deg,	R =   90.000 deg
};
P[445]{
   GP1:
	UF : 0, UT : 6,		CONFIG : 'N U T, 0, 0, 0',
	X =  290.233  mm,	Y =   -283.795  mm,	Z =   -269.340  mm,
	W =  90.000 deg,	P =   0.000 deg,	R =   90.000 deg
};
P[446]{
   GP1:
	UF : 0, UT : 6,		CONFIG : 'N U T, 0, 0, 0',
	X =  289.068  mm,	Y =   -281.751  mm,	Z =   -269.250  mm,
	W =  90.000 deg,	P =   0.000 deg,	R =   90.000 deg
};
P[447]{
   GP1:
	UF : 0, UT : 6,		CONFIG : 'N U T, 0, 0, 0',
	X =  287.816  mm,	Y =   -279.579  mm,	Z =   -269.238  mm,
	W =  90.000 deg,	P =   0.000 deg,	R =   90.000 deg
};
P[448]{
   GP1:
	UF : 0, UT : 6,		CONFIG : 'N U T, 0, 0, 0',
	X =  286.082  mm,	Y =   -276.612  mm,	Z =   -269.363  mm,
	W =  90.000 deg,	P =   0.000 deg,	R =   90.000 deg
};
P[449]{
   GP1:
	UF : 0, UT : 6,		CONFIG : 'N U T, 0, 0, 0',
	X =  285.518  mm,	Y =   -275.653  mm,	Z =   -269.425  mm,
	W =  90.000 deg,	P =   0.000 deg,	R =   90.000 deg
};
P[450]{
   GP1:
	UF : 0, UT : 6,		CONFIG : 'N U T, 0, 0, 0',
	X =  284.424  mm,	Y =   -273.638  mm,	Z =   -268.998  mm,
	W =  90.000 deg,	P =   0.000 deg,	R =   90.000 deg
};
P[451]{
   GP1:
	UF : 0, UT : 6,		CONFIG : 'N U T, 0, 0, 0',
	X =  283.009  mm,	Y =   -271.292  mm,	Z =   -269.371  mm,
	W =  90.000 deg,	P =   0.000 deg,	R =   90.000 deg
};
P[452]{
   GP1:
	UF : 0, UT : 6,		CONFIG : 'N U T, 0, 0, 0',
	X =  281.517  mm,	Y =   -268.667  mm,	Z =   -269.225  mm,
	W =  90.000 deg,	P =   0.000 deg,	R =   90.000 deg
};
P[453]{
   GP1:
	UF : 0, UT : 6,		CONFIG : 'N U T, 0, 0, 0',
	X =  280.889  mm,	Y =   -267.633  mm,	Z =   -269.417  mm,
	W =  90.000 deg,	P =   0.000 deg,	R =   90.000 deg
};
P[454]{
   GP1:
	UF : 0, UT : 6,		CONFIG : 'N U T, 0, 0, 0',
	X =  280.172  mm,	Y =   -266.380  mm,	Z =   -269.376  mm,
	W =  90.000 deg,	P =   0.000 deg,	R =   90.000 deg
};
P[455]{
   GP1:
	UF : 0, UT : 6,		CONFIG : 'N U T, 0, 0, 0',
	X =  278.074  mm,	Y =   -262.670  mm,	Z =   -269.106  mm,
	W =  90.000 deg,	P =   0.000 deg,	R =   90.000 deg
};
P[456]{
   GP1:
	UF : 0, UT : 6,		CONFIG : 'N U T, 0, 0, 0',
	X =  277.372  mm,	Y =   -261.550  mm,	Z =   -269.447  mm,
	W =  90.000 deg,	P =   0.000 deg,	R =   90.000 deg
};
P[457]{
   GP1:
	UF : 0, UT : 6,		CONFIG : 'N U T, 0, 0, 0',
	X =  276.591  mm,	Y =   -260.143  mm,	Z =   -269.248  mm,
	W =  90.000 deg,	P =   0.000 deg,	R =   90.000 deg
};
P[458]{
   GP1:
	UF : 0, UT : 6,		CONFIG : 'N U T, 0, 0, 0',
	X =  276.056  mm,	Y =   -259.202  mm,	Z =   -269.195  mm,
	W =  90.000 deg,	P =   0.000 deg,	R =   90.000 deg
};
P[459]{
   GP1:
	UF : 0, UT : 6,		CONFIG : 'N U T, 0, 0, 0',
	X =  275.303  mm,	Y =   -257.936  mm,	Z =   -269.336  mm,
	W =  90.000 deg,	P =   0.000 deg,	R =   90.000 deg
};
P[460]{
   GP1:
	UF : 0, UT : 6,		CONFIG : 'N U T, 0, 0, 0',
	X =  274.692  mm,	Y =   -256.877  mm,	Z =   -269.334  mm,
	W =  90.000 deg,	P =   0.000 deg,	R =   90.000 deg
};
P[461]{
   GP1:
	UF : 0, UT : 6,		CONFIG : 'N U T, 0, 0, 0',
	X =  274.215  mm,	Y =   -256.044  mm,	Z =   -269.313  mm,
	W =  90.000 deg,	P =   0.000 deg,	R =   90.000 deg
};
P[462]{
   GP1:
	UF : 0, UT : 6,		CONFIG : 'N U T, 0, 0, 0',
	X =  273.283  mm,	Y =   -254.473  mm,	Z =   -269.459  mm,
	W =  90.000 deg,	P =   0.000 deg,	R =   90.000 deg
};
P[463]{
   GP1:
	UF : 0, UT : 6,		CONFIG : 'N U T, 0, 0, 0',
	X =  272.682  mm,	Y =   -253.387  mm,	Z =   -269.304  mm,
	W =  90.000 deg,	P =   0.000 deg,	R =   90.000 deg
};
P[464]{
   GP1:
	UF : 0, UT : 6,		CONFIG : 'N U T, 0, 0, 0',
	X =  270.983  mm,	Y =   -250.450  mm,	Z =   -269.320  mm,
	W =  90.000 deg,	P =   0.000 deg,	R =   90.000 deg
};
P[465]{
   GP1:
	UF : 0, UT : 6,		CONFIG : 'N U T, 0, 0, 0',
	X =  269.515  mm,	Y =   -247.856  mm,	Z =   -269.142  mm,
	W =  90.000 deg,	P =   0.000 deg,	R =   90.000 deg
};
P[466]{
   GP1:
	UF : 0, UT : 6,		CONFIG : 'N U T, 0, 0, 0',
	X =  268.644  mm,	Y =   -246.392  mm,	Z =   -269.297  mm,
	W =  90.000 deg,	P =   0.000 deg,	R =   90.000 deg
};
P[467]{
   GP1:
	UF : 0, UT : 6,		CONFIG : 'N U T, 0, 0, 0',
	X =  268.233  mm,	Y =   -245.615  mm,	Z =   -269.070  mm,
	W =  90.000 deg,	P =   0.000 deg,	R =   90.000 deg
};
P[468]{
   GP1:
	UF : 0, UT : 6,		CONFIG : 'N U T, 0, 0, 0',
	X =  267.785  mm,	Y =   -244.943  mm,	Z =   -269.435  mm,
	W =  90.000 deg,	P =   0.000 deg,	R =   90.000 deg
};
P[469]{
   GP1:
	UF : 0, UT : 6,		CONFIG : 'N U T, 0, 0, 0',
	X =  266.800  mm,	Y =   -243.206  mm,	Z =   -269.320  mm,
	W =  90.000 deg,	P =   0.000 deg,	R =   90.000 deg
};
P[470]{
   GP1:
	UF : 0, UT : 6,		CONFIG : 'N U T, 0, 0, 0',
	X =  266.003  mm,	Y =   -241.769  mm,	Z =   -269.125  mm,
	W =  90.000 deg,	P =   0.000 deg,	R =   90.000 deg
};
P[471]{
   GP1:
	UF : 0, UT : 6,		CONFIG : 'N U T, 0, 0, 0',
	X =  264.588  mm,	Y =   -239.391  mm,	Z =   -269.380  mm,
	W =  90.000 deg,	P =   0.000 deg,	R =   90.000 deg
};
P[472]{
   GP1:
	UF : 0, UT : 6,		CONFIG : 'N U T, 0, 0, 0',
	X =  263.973  mm,	Y =   -238.230  mm,	Z =   -269.039  mm,
	W =  90.000 deg,	P =   0.000 deg,	R =   90.000 deg
};
P[473]{
   GP1:
	UF : 0, UT : 6,		CONFIG : 'N U T, 0, 0, 0',
	X =  263.106  mm,	Y =   -236.800  mm,	Z =   -269.294  mm,
	W =  90.000 deg,	P =   0.000 deg,	R =   90.000 deg
};
P[474]{
   GP1:
	UF : 0, UT : 6,		CONFIG : 'N U T, 0, 0, 0',
	X =  262.611  mm,	Y =   -235.935  mm,	Z =   -269.271  mm,
	W =  90.000 deg,	P =   0.000 deg,	R =   90.000 deg
};
P[475]{
   GP1:
	UF : 0, UT : 6,		CONFIG : 'N U T, 0, 0, 0',
	X =  262.122  mm,	Y =   -235.078  mm,	Z =   -269.229  mm,
	W =  90.000 deg,	P =   0.000 deg,	R =   90.000 deg
};
P[476]{
   GP1:
	UF : 0, UT : 6,		CONFIG : 'N U T, 0, 0, 0',
	X =  261.222  mm,	Y =   -233.580  mm,	Z =   -269.453  mm,
	W =  90.000 deg,	P =   0.000 deg,	R =   90.000 deg
};
P[477]{
   GP1:
	UF : 0, UT : 6,		CONFIG : 'N U T, 0, 0, 0',
	X =  260.745  mm,	Y =   -232.744  mm,	Z =   -269.416  mm,
	W =  90.000 deg,	P =   0.000 deg,	R =   90.000 deg
};
P[478]{
   GP1:
	UF : 0, UT : 6,		CONFIG : 'N U T, 0, 0, 0',
	X =  260.048  mm,	Y =   -231.491  mm,	Z =   -269.248  mm,
	W =  90.000 deg,	P =   0.000 deg,	R =   90.000 deg
};
P[479]{
   GP1:
	UF : 0, UT : 6,		CONFIG : 'N U T, 0, 0, 0',
	X =  258.853  mm,	Y =   -229.454  mm,	Z =   -269.364  mm,
	W =  90.000 deg,	P =   0.000 deg,	R =   90.000 deg
};
P[480]{
   GP1:
	UF : 0, UT : 6,		CONFIG : 'N U T, 0, 0, 0',
	X =  258.158  mm,	Y =   -228.169  mm,	Z =   -269.077  mm,
	W =  90.000 deg,	P =   0.000 deg,	R =   90.000 deg
};
P[481]{
   GP1:
	UF : 0, UT : 6,		CONFIG : 'N U T, 0, 0, 0',
	X =  257.564  mm,	Y =   -227.189  mm,	Z =   -269.249  mm,
	W =  90.000 deg,	P =   0.000 deg,	R =   90.000 deg
};
P[482]{
   GP1:
	UF : 0, UT : 6,		CONFIG : 'N U T, 0, 0, 0',
	X =  256.597  mm,	Y =   -225.551  mm,	Z =   -269.387  mm,
	W =  90.000 deg,	P =   0.000 deg,	R =   90.000 deg
};
P[483]{
   GP1:
	UF : 0, UT : 6,		CONFIG : 'N U T, 0, 0, 0',
	X =  255.233  mm,	Y =   -223.198  mm,	Z =   -269.413  mm,
	W =  90.000 deg,	P =   0.000 deg,	R =   90.000 deg
};
P[484]{
   GP1:
	UF : 0, UT : 6,		CONFIG : 'N U T, 0, 0, 0',
	X =  254.799  mm,	Y =   -222.427  mm,	Z =   -269.351  mm,
	W =  90.000 deg,	P =   0.000 deg,	R =   90.000 deg
};
P[485]{
   GP1:
	UF : 0, UT : 6,		CONFIG : 'N U T, 0, 0, 0',
	X =  254.371  mm,	Y =   -221.699  mm,	Z =   -269.393  mm,
	W =  90.000 deg,	P =   0.000 deg,	R =   90.000 deg
};
P[486]{
   GP1:
	UF : 0, UT : 6,		CONFIG : 'N U T, 0, 0, 0',
	X =  253.608  mm,	Y =   -220.582  mm,	Z =   -269.247  mm,
	W =  90.000 deg,	P =   0.000 deg,	R =   90.000 deg
};
P[487]{
   GP1:
	UF : 0, UT : 6,		CONFIG : 'N U T, 0, 0, 0',
	X =  252.866  mm,	Y =   -219.951  mm,	Z =   -269.187  mm,
	W =  90.000 deg,	P =   0.000 deg,	R =   90.000 deg
};
P[488]{
   GP1:
	UF : 0, UT : 6,		CONFIG : 'N U T, 0, 0, 0',
	X =  251.916  mm,	Y =   -219.535  mm,	Z =   -269.395  mm,
	W =  90.000 deg,	P =   0.000 deg,	R =   90.000 deg
};
P[489]{
   GP1:
	UF : 0, UT : 6,		CONFIG : 'N U T, 0, 0, 0',
	X =  250.646  mm,	Y =   -219.296  mm,	Z =   -269.367  mm,
	W =  90.000 deg,	P =   0.000 deg,	R =   90.000 deg
};
P[490]{
   GP1:
	UF : 0, UT : 6,		CONFIG : 'N U T, 0, 0, 0',
	X =  248.976  mm,	Y =   -219.678  mm,	Z =   -269.395  mm,
	W =  90.000 deg,	P =   0.000 deg,	R =   90.000 deg
};
P[491]{
   GP1:
	UF : 0, UT : 6,		CONFIG : 'N U T, 0, 0, 0',
	X =  248.305  mm,	Y =   -219.969  mm,	Z =   -269.218  mm,
	W =  90.000 deg,	P =   0.000 deg,	R =   90.000 deg
};
P[492]{
   GP1:
	UF : 0, UT : 6,		CONFIG : 'N U T, 0, 0, 0',
	X =  247.527  mm,	Y =   -220.441  mm,	Z =   -269.355  mm,
	W =  90.000 deg,	P =   0.000 deg,	R =   90.000 deg
};
P[493]{
   GP1:
	UF : 0, UT : 6,		CONFIG : 'N U T, 0, 0, 0',
	X =  245.472  mm,	Y =   -221.641  mm,	Z =   -269.439  mm,
	W =  90.000 deg,	P =   0.000 deg,	R =   90.000 deg
};
P[494]{
   GP1:
	UF : 0, UT : 6,		CONFIG : 'N U T, 0, 0, 0',
	X =  242.354  mm,	Y =   -223.369  mm,	Z =   -268.992  mm,
	W =  90.000 deg,	P =   0.000 deg,	R =   90.000 deg
};
P[495]{
   GP1:
	UF : 0, UT : 6,		CONFIG : 'N U T, 0, 0, 0',
	X =  240.330  mm,	Y =   -224.564  mm,	Z =   -269.161  mm,
	W =  90.000 deg,	P =   0.000 deg,	R =   90.000 deg
};
P[496]{
   GP1:
	UF : 0, UT : 6,		CONFIG : 'N U T, 0, 0, 0',
	X =  239.568  mm,	Y =   -225.047  mm,	Z =   -269.424  mm,
	W =  90.000 deg,	P =   0.000 deg,	R =   90.000 deg
};
P[497]{
   GP1:
	UF : 0, UT : 6,		CONFIG : 'N U T, 0, 0, 0',
	X =  238.745  mm,	Y =   -225.510  mm,	Z =   -269.347  mm,
	W =  90.000 deg,	P =   0.000 deg,	R =   90.000 deg
};
P[498]{
   GP1:
	UF : 0, UT : 6,		CONFIG : 'N U T, 0, 0, 0',
	X =  236.609  mm,	Y =   -226.761  mm,	Z =   -269.454  mm,
	W =  90.000 deg,	P =   0.000 deg,	R =   90.000 deg
};
P[499]{
   GP1:
	UF : 0, UT : 6,		CONFIG : 'N U T, 0, 0, 0',
	X =  234.921  mm,	Y =   -227.708  mm,	Z =   -269.287  mm,
	W =  90.000 deg,	P =   0.000 deg,	R =   90.000 deg
};
P[500]{
   GP1:
	UF : 0, UT : 6,		CONFIG : 'N U T, 0, 0, 0',
	X =  233.983  mm,	Y =   -228.234  mm,	Z =   -269.191  mm,
	W =  90.000 deg,	P =   0.000 deg,	R =   90.000 deg
};
P[501]{
   GP1:
	UF : 0, UT : 6,		CONFIG : 'N U T, 0, 0, 0',
	X =  233.045  mm,	Y =   -228.805  mm,	Z =   -269.370  mm,
	W =  90.000 deg,	P =   0.000 deg,	R =   90.000 deg
};
P[502]{
   GP1:
	UF : 0, UT : 6,		CONFIG : 'N U T, 0, 0, 0',
	X =  231.716  mm,	Y =   -229.562  mm,	Z =   -269.311  mm,
	W =  90.000 deg,	P =   0.000 deg,	R =   90.000 deg
};
P[503]{
   GP1:
	UF : 0, UT : 6,		CONFIG : 'N U T, 0, 0, 0',
	X =  230.980  mm,	Y =   -229.987  mm,	Z =   -269.311  mm,
	W =  90.000 deg,	P =   0.000 deg,	R =   90.000 deg
};
P[504]{
   GP1:
	UF : 0, UT : 6,		CONFIG : 'N U T, 0, 0, 0',
	X =  230.016  mm,	Y =   -230.558  mm,	Z =   -269.393  mm,
	W =  90.000 deg,	P =   0.000 deg,	R =   90.000 deg
};
P[505]{
   GP1:
	UF : 0, UT : 6,		CONFIG : 'N U T, 0, 0, 0',
	X =  229.101  mm,	Y =   -231.049  mm,	Z =   -269.165  mm,
	W =  90.000 deg,	P =   0.000 deg,	R =   90.000 deg
};
P[506]{
   GP1:
	UF : 0, UT : 6,		CONFIG : 'N U T, 0, 0, 0',
	X =  228.238  mm,	Y =   -231.539  mm,	Z =   -269.120  mm,
	W =  90.000 deg,	P =   0.000 deg,	R =   90.000 deg
};
P[507]{
   GP1:
	UF : 0, UT : 6,		CONFIG : 'N U T, 0, 0, 0',
	X =  226.211  mm,	Y =   -232.725  mm,	Z =   -269.211  mm,
	W =  90.000 deg,	P =   0.000 deg,	R =   90.000 deg
};
P[508]{
   GP1:
	UF : 0, UT : 6,		CONFIG : 'N U T, 0, 0, 0',
	X =  224.148  mm,	Y =   -233.950  mm,	Z =   -269.422  mm,
	W =  90.000 deg,	P =   0.000 deg,	R =   90.000 deg
};
P[509]{
   GP1:
	UF : 0, UT : 6,		CONFIG : 'N U T, 0, 0, 0',
	X =  222.935  mm,	Y =   -234.606  mm,	Z =   -269.146  mm,
	W =  90.000 deg,	P =   0.000 deg,	R =   90.000 deg
};
P[510]{
   GP1:
	UF : 0, UT : 6,		CONFIG : 'N U T, 0, 0, 0',
	X =  220.984  mm,	Y =   -235.705  mm,	Z =   -268.974  mm,
	W =  90.000 deg,	P =   0.000 deg,	R =   90.000 deg
};
P[511]{
   GP1:
	UF : 0, UT : 6,		CONFIG : 'N U T, 0, 0, 0',
	X =  220.319  mm,	Y =   -236.090  mm,	Z =   -268.988  mm,
	W =  90.000 deg,	P =   0.000 deg,	R =   90.000 deg
};
P[512]{
   GP1:
	UF : 0, UT : 6,		CONFIG : 'N U T, 0, 0, 0',
	X =  218.806  mm,	Y =   -237.027  mm,	Z =   -269.377  mm,
	W =  90.000 deg,	P =   0.000 deg,	R =   90.000 deg
};
P[513]{
   GP1:
	UF : 0, UT : 6,		CONFIG : 'N U T, 0, 0, 0',
	X =  216.657  mm,	Y =   -238.275  mm,	Z =   -269.423  mm,
	W =  90.000 deg,	P =   0.000 deg,	R =   90.000 deg
};
P[514]{
   GP1:
	UF : 0, UT : 6,		CONFIG : 'N U T, 0, 0, 0',
	X =  215.448  mm,	Y =   -238.976  mm,	Z =   -269.437  mm,
	W =  90.000 deg,	P =   0.000 deg,	R =   90.000 deg
};
P[515]{
   GP1:
	UF : 0, UT : 6,		CONFIG : 'N U T, 0, 0, 0',
	X =  214.863  mm,	Y =   -239.301  mm,	Z =   -269.358  mm,
	W =  90.000 deg,	P =   0.000 deg,	R =   90.000 deg
};
P[516]{
   GP1:
	UF : 0, UT : 6,		CONFIG : 'N U T, 0, 0, 0',
	X =  214.149  mm,	Y =   -239.678  mm,	Z =   -269.142  mm,
	W =  90.000 deg,	P =   0.000 deg,	R =   90.000 deg
};
P[517]{
   GP1:
	UF : 0, UT : 6,		CONFIG : 'N U T, 0, 0, 0',
	X =  210.617  mm,	Y =   -241.725  mm,	Z =   -269.194  mm,
	W =  90.000 deg,	P =   0.000 deg,	R =   90.000 deg
};
P[518]{
   GP1:
	UF : 0, UT : 6,		CONFIG : 'N U T, 0, 0, 0',
	X =  209.915  mm,	Y =   -242.172  mm,	Z =   -269.448  mm,
	W =  90.000 deg,	P =   0.000 deg,	R =   90.000 deg
};
P[519]{
   GP1:
	UF : 0, UT : 6,		CONFIG : 'N U T, 0, 0, 0',
	X =  207.694  mm,	Y =   -243.410  mm,	Z =   -269.172  mm,
	W =  90.000 deg,	P =   0.000 deg,	R =   90.000 deg
};
P[520]{
   GP1:
	UF : 0, UT : 6,		CONFIG : 'N U T, 0, 0, 0',
	X =  205.844  mm,	Y =   -244.500  mm,	Z =   -269.311  mm,
	W =  90.000 deg,	P =   0.000 deg,	R =   90.000 deg
};
P[521]{
   GP1:
	UF : 0, UT : 6,		CONFIG : 'N U T, 0, 0, 0',
	X =  205.020  mm,	Y =   -244.957  mm,	Z =   -269.191  mm,
	W =  90.000 deg,	P =   0.000 deg,	R =   90.000 deg
};
P[522]{
   GP1:
	UF : 0, UT : 6,		CONFIG : 'N U T, 0, 0, 0',
	X =  203.618  mm,	Y =   -245.797  mm,	Z =   -269.374  mm,
	W =  90.000 deg,	P =   0.000 deg,	R =   90.000 deg
};
P[523]{
   GP1:
	UF : 0, UT : 6,		CONFIG : 'N U T, 0, 0, 0',
	X =  202.667  mm,	Y =   -246.317  mm,	Z =   -269.196  mm,
	W =  90.000 deg,	P =   0.000 deg,	R =   90.000 deg
};
P[524]{
   GP1:
	UF : 0, UT : 6,		CONFIG : 'N U T, 0, 0, 0',
	X =  202.038  mm,	Y =   -246.642  mm,	Z =   -268.967  mm,
	W =  90.000 deg,	P =   0.000 deg,	R =   90.000 deg
};
P[525]{
   GP1:
	UF : 0, UT : 6,		CONFIG : 'N U T, 0, 0, 0',
	X =  201.083  mm,	Y =   -247.231  mm,	Z =   -269.200  mm,
	W =  90.000 deg,	P =   0.000 deg,	R =   90.000 deg
};
P[526]{
   GP1:
	UF : 0, UT : 6,		CONFIG : 'N U T, 0, 0, 0',
	X =  200.270  mm,	Y =   -247.719  mm,	Z =   -269.310  mm,
	W =  90.000 deg,	P =   0.000 deg,	R =   90.000 deg
};
P[527]{
   GP1:
	UF : 0, UT : 6,		CONFIG : 'N U T, 0, 0, 0',
	X =  198.958  mm,	Y =   -248.463  mm,	Z =   -269.224  mm,
	W =  90.000 deg,	P =   0.000 deg,	R =   90.000 deg
};
P[528]{
   GP1:
	UF : 0, UT : 6,		CONFIG : 'N U T, 0, 0, 0',
	X =  197.991  mm,	Y =   -249.007  mm,	Z =   -269.138  mm,
	W =  90.000 deg,	P =   0.000 deg,	R =   90.000 deg
};
P[529]{
   GP1:
	UF : 0, UT : 6,		CONFIG : 'N U T, 0, 0, 0',
	X =  195.934  mm,	Y =   -250.219  mm,	Z =   -269.290  mm,
	W =  90.000 deg,	P =   0.000 deg,	R =   90.000 deg
};
P[530]{
   GP1:
	UF : 0, UT : 6,		CONFIG : 'N U T, 0, 0, 0',
	X =  193.812  mm,	Y =   -251.439  mm,	Z =   -269.255  mm,
	W =  90.000 deg,	P =   0.000 deg,	R =   90.000 deg
};
P[531]{
   GP1:
	UF : 0, UT : 6,		CONFIG : 'N U T, 0, 0, 0',
	X =  192.626  mm,	Y =   -252.132  mm,	Z =   -269.307  mm,
	W =  90.000 deg,	P =   0.000 deg,	R =   90.000 deg
};
P[532]{
   GP1:
	UF : 0, UT : 6,		CONFIG : 'N U T, 0, 0, 0',
	X =  190.008  mm,	Y =   -253.633  mm,	Z =   -269.244  mm,
	W =  90.000 deg,	P =   0.000 deg,	R =   90.000 deg
};
P[533]{
   GP1:
	UF : 0, UT : 6,		CONFIG : 'N U T, 0, 0, 0',
	X =  189.231  mm,	Y =   -254.051  mm,	Z =   -269.052  mm,
	W =  90.000 deg,	P =   0.000 deg,	R =   90.000 deg
};
P[534]{
   GP1:
	UF : 0, UT : 6,		CONFIG : 'N U T, 0, 0, 0',
	X =  187.379  mm,	Y =   -255.177  mm,	Z =   -269.401  mm,
	W =  90.000 deg,	P =   0.000 deg,	R =   90.000 deg
};
P[535]{
   GP1:
	UF : 0, UT : 6,		CONFIG : 'N U T, 0, 0, 0',
	X =  184.339  mm,	Y =   -256.874  mm,	Z =   -269.041  mm,
	W =  90.000 deg,	P =   0.000 deg,	R =   90.000 deg
};
P[536]{
   GP1:
	UF : 0, UT : 6,		CONFIG : 'N U T, 0, 0, 0',
	X =  182.678  mm,	Y =   -257.882  mm,	Z =   -269.342  mm,
	W =  90.000 deg,	P =   0.000 deg,	R =   90.000 deg
};
P[537]{
   GP1:
	UF : 0, UT : 6,		CONFIG : 'N U T, 0, 0, 0',
	X =  179.645  mm,	Y =   -259.602  mm,	Z =   -269.153  mm,
	W =  90.000 deg,	P =   0.000 deg,	R =   90.000 deg
};
P[538]{
   GP1:
	UF : 0, UT : 6,		CONFIG : 'N U T, 0, 0, 0',
	X =  178.008  mm,	Y =   -260.585  mm,	Z =   -269.387  mm,
	W =  90.000 deg,	P =   0.000 deg,	R =   90.000 deg
};
P[539]{
   GP1:
	UF : 0, UT : 6,		CONFIG : 'N U T, 0, 0, 0',
	X =  177.073  mm,	Y =   -261.062  mm,	Z =   -269.000  mm,
	W =  90.000 deg,	P =   0.000 deg,	R =   90.000 deg
};
P[540]{
   GP1:
	UF : 0, UT : 6,		CONFIG : 'N U T, 0, 0, 0',
	X =  176.501  mm,	Y =   -261.415  mm,	Z =   -269.142  mm,
	W =  90.000 deg,	P =   0.000 deg,	R =   90.000 deg
};
P[541]{
   GP1:
	UF : 0, UT : 6,		CONFIG : 'N U T, 0, 0, 0',
	X =  173.941  mm,	Y =   -262.886  mm,	Z =   -269.090  mm,
	W =  90.000 deg,	P =   0.000 deg,	R =   90.000 deg
};
P[542]{
   GP1:
	UF : 0, UT : 6,		CONFIG : 'N U T, 0, 0, 0',
	X =  173.189  mm,	Y =   -263.357  mm,	Z =   -269.322  mm,
	W =  90.000 deg,	P =   0.000 deg,	R =   90.000 deg
};
P[543]{
   GP1:
	UF : 0, UT : 6,		CONFIG : 'N U T, 0, 0, 0',
	X =  166.967  mm,	Y =   -266.950  mm,	Z =   -269.325  mm,
	W =  90.000 deg,	P =   0.000 deg,	R =   90.000 deg
};
P[544]{
   GP1:
	UF : 0, UT : 6,		CONFIG : 'N U T, 0, 0, 0',
	X =  166.187  mm,	Y =   -267.418  mm,	Z =   -269.431  mm,
	W =  90.000 deg,	P =   0.000 deg,	R =   90.000 deg
};
P[545]{
   GP1:
	UF : 0, UT : 6,		CONFIG : 'N U T, 0, 0, 0',
	X =  164.667  mm,	Y =   -268.286  mm,	Z =   -269.370  mm,
	W =  90.000 deg,	P =   0.000 deg,	R =   90.000 deg
};
P[546]{
   GP1:
	UF : 0, UT : 6,		CONFIG : 'N U T, 0, 0, 0',
	X =  163.818  mm,	Y =   -268.786  mm,	Z =   -269.435  mm,
	W =  90.000 deg,	P =   0.000 deg,	R =   90.000 deg
};
P[547]{
   GP1:
	UF : 0, UT : 6,		CONFIG : 'N U T, 0, 0, 0',
	X =  163.039  mm,	Y =   -269.213  mm,	Z =   -269.299  mm,
	W =  90.000 deg,	P =   0.000 deg,	R =   90.000 deg
};
P[548]{
   GP1:
	UF : 0, UT : 6,		CONFIG : 'N U T, 0, 0, 0',
	X =  160.665  mm,	Y =   -270.555  mm,	Z =   -269.119  mm,
	W =  90.000 deg,	P =   0.000 deg,	R =   90.000 deg
};
P[549]{
   GP1:
	UF : 0, UT : 6,		CONFIG : 'N U T, 0, 0, 0',
	X =  159.820  mm,	Y =   -271.049  mm,	Z =   -269.157  mm,
	W =  90.000 deg,	P =   0.000 deg,	R =   90.000 deg
};
P[550]{
   GP1:
	UF : 0, UT : 6,		CONFIG : 'N U T, 0, 0, 0',
	X =  158.627  mm,	Y =   -271.754  mm,	Z =   -269.252  mm,
	W =  90.000 deg,	P =   0.000 deg,	R =   90.000 deg
};
P[551]{
   GP1:
	UF : 0, UT : 6,		CONFIG : 'N U T, 0, 0, 0',
	X =  157.889  mm,	Y =   -272.194  mm,	Z =   -269.333  mm,
	W =  90.000 deg,	P =   0.000 deg,	R =   90.000 deg
};
P[552]{
   GP1:
	UF : 0, UT : 6,		CONFIG : 'N U T, 0, 0, 0',
	X =  157.371  mm,	Y =   -272.498  mm,	Z =   -269.373  mm,
	W =  90.000 deg,	P =   0.000 deg,	R =   90.000 deg
};
P[553]{
   GP1:
	UF : 0, UT : 6,		CONFIG : 'N U T, 0, 0, 0',
	X =  156.537  mm,	Y =   -272.981  mm,	Z =   -269.373  mm,
	W =  90.000 deg,	P =   0.000 deg,	R =   90.000 deg
};
P[554]{
   GP1:
	UF : 0, UT : 6,		CONFIG : 'N U T, 0, 0, 0',
	X =  153.147  mm,	Y =   -274.907  mm,	Z =   -269.184  mm,
	W =  90.000 deg,	P =   0.000 deg,	R =   90.000 deg
};
P[555]{
   GP1:
	UF : 0, UT : 6,		CONFIG : 'N U T, 0, 0, 0',
	X =  150.987  mm,	Y =   -275.250  mm,	Z =   -263.616  mm,
	W =  90.000 deg,	P =   0.000 deg,	R =   90.000 deg
};
P[556]{
   GP1:
	UF : 0, UT : 6,		CONFIG : 'N U T, 0, 0, 0',
	X =  149.970  mm,	Y =   -275.806  mm,	Z =   -263.422  mm,
	W =  90.000 deg,	P =   0.000 deg,	R =   90.000 deg
};
P[557]{
   GP1:
	UF : 0, UT : 6,		CONFIG : 'N U T, 0, 0, 0',
	X =  149.146  mm,	Y =   -276.315  mm,	Z =   -263.624  mm,
	W =  90.000 deg,	P =   0.000 deg,	R =   90.000 deg
};
P[558]{
   GP1:
	UF : 0, UT : 6,		CONFIG : 'N U T, 0, 0, 0',
	X =  147.127  mm,	Y =   -277.482  mm,	Z =   -263.635  mm,
	W =  90.000 deg,	P =   0.000 deg,	R =   90.000 deg
};
P[559]{
   GP1:
	UF : 0, UT : 6,		CONFIG : 'N U T, 0, 0, 0',
	X =  146.268  mm,	Y =   -278.019  mm,	Z =   -263.888  mm,
	W =  90.000 deg,	P =   0.000 deg,	R =   90.000 deg
};
P[560]{
   GP1:
	UF : 0, UT : 6,		CONFIG : 'N U T, 0, 0, 0',
	X =  143.187  mm,	Y =   -279.752  mm,	Z =   -263.598  mm,
	W =  90.000 deg,	P =   0.000 deg,	R =   90.000 deg
};
P[561]{
   GP1:
	UF : 0, UT : 6,		CONFIG : 'N U T, 0, 0, 0',
	X =  142.096  mm,	Y =   -280.391  mm,	Z =   -263.660  mm,
	W =  90.000 deg,	P =   0.000 deg,	R =   90.000 deg
};
P[562]{
   GP1:
	UF : 0, UT : 6,		CONFIG : 'N U T, 0, 0, 0',
	X =  141.418  mm,	Y =   -280.757  mm,	Z =   -263.504  mm,
	W =  90.000 deg,	P =   0.000 deg,	R =   90.000 deg
};
P[563]{
   GP1:
	UF : 0, UT : 6,		CONFIG : 'N U T, 0, 0, 0',
	X =  140.096  mm,	Y =   -281.542  mm,	Z =   -263.638  mm,
	W =  90.000 deg,	P =   0.000 deg,	R =   90.000 deg
};
P[564]{
   GP1:
	UF : 0, UT : 6,		CONFIG : 'N U T, 0, 0, 0',
	X =  138.110  mm,	Y =   -282.695  mm,	Z =   -263.670  mm,
	W =  90.000 deg,	P =   0.000 deg,	R =   90.000 deg
};
P[565]{
   GP1:
	UF : 0, UT : 6,		CONFIG : 'N U T, 0, 0, 0',
	X =  133.874  mm,	Y =   -285.111  mm,	Z =   -263.488  mm,
	W =  90.000 deg,	P =   0.000 deg,	R =   90.000 deg
};
P[566]{
   GP1:
	UF : 0, UT : 6,		CONFIG : 'N U T, 0, 0, 0',
	X =  133.002  mm,	Y =   -285.635  mm,	Z =   -263.617  mm,
	W =  90.000 deg,	P =   0.000 deg,	R =   90.000 deg
};
P[567]{
   GP1:
	UF : 0, UT : 6,		CONFIG : 'N U T, 0, 0, 0',
	X =  132.077  mm,	Y =   -286.205  mm,	Z =   -263.838  mm,
	W =  90.000 deg,	P =   0.000 deg,	R =   90.000 deg
};
P[568]{
   GP1:
	UF : 0, UT : 6,		CONFIG : 'N U T, 0, 0, 0',
	X =  131.388  mm,	Y =   -286.535  mm,	Z =   -263.425  mm,
	W =  90.000 deg,	P =   0.000 deg,	R =   90.000 deg
};
P[569]{
   GP1:
	UF : 0, UT : 6,		CONFIG : 'N U T, 0, 0, 0',
	X =  128.970  mm,	Y =   -287.992  mm,	Z =   -263.800  mm,
	W =  90.000 deg,	P =   0.000 deg,	R =   90.000 deg
};
P[570]{
   GP1:
	UF : 0, UT : 6,		CONFIG : 'N U T, 0, 0, 0',
	X =  127.248  mm,	Y =   -288.956  mm,	Z =   -263.612  mm,
	W =  90.000 deg,	P =   0.000 deg,	R =   90.000 deg
};
P[571]{
   GP1:
	UF : 0, UT : 6,		CONFIG : 'N U T, 0, 0, 0',
	X =  126.251  mm,	Y =   -289.551  mm,	Z =   -263.723  mm,
	W =  90.000 deg,	P =   0.000 deg,	R =   90.000 deg
};
P[572]{
   GP1:
	UF : 0, UT : 6,		CONFIG : 'N U T, 0, 0, 0',
	X =  125.353  mm,	Y =   -290.038  mm,	Z =   -263.536  mm,
	W =  90.000 deg,	P =   0.000 deg,	R =   90.000 deg
};
P[573]{
   GP1:
	UF : 0, UT : 6,		CONFIG : 'N U T, 0, 0, 0',
	X =  124.745  mm,	Y =   -290.431  mm,	Z =   -263.788  mm,
	W =  90.000 deg,	P =   0.000 deg,	R =   90.000 deg
};
P[574]{
   GP1:
	UF : 0, UT : 6,		CONFIG : 'N U T, 0, 0, 0',
	X =  123.520  mm,	Y =   -291.089  mm,	Z =   -263.491  mm,
	W =  90.000 deg,	P =   0.000 deg,	R =   90.000 deg
};
P[575]{
   GP1:
	UF : 0, UT : 6,		CONFIG : 'N U T, 0, 0, 0',
	X =  121.749  mm,	Y =   -292.118  mm,	Z =   -263.527  mm,
	W =  90.000 deg,	P =   0.000 deg,	R =   90.000 deg
};
P[576]{
   GP1:
	UF : 0, UT : 6,		CONFIG : 'N U T, 0, 0, 0',
	X =  120.889  mm,	Y =   -292.641  mm,	Z =   -263.690  mm,
	W =  90.000 deg,	P =   0.000 deg,	R =   90.000 deg
};
P[577]{
   GP1:
	UF : 0, UT : 6,		CONFIG : 'N U T, 0, 0, 0',
	X =  119.785  mm,	Y =   -293.271  mm,	Z =   -263.645  mm,
	W =  90.000 deg,	P =   0.000 deg,	R =   90.000 deg
};
P[578]{
   GP1:
	UF : 0, UT : 6,		CONFIG : 'N U T, 0, 0, 0',
	X =  117.735  mm,	Y =   -294.424  mm,	Z =   -263.458  mm,
	W =  90.000 deg,	P =   0.000 deg,	R =   90.000 deg
};
P[579]{
   GP1:
	UF : 0, UT : 6,		CONFIG : 'N U T, 0, 0, 0',
	X =  115.881  mm,	Y =   -295.569  mm,	Z =   -263.914  mm,
	W =  90.000 deg,	P =   0.000 deg,	R =   90.000 deg
};
P[580]{
   GP1:
	UF : 0, UT : 6,		CONFIG : 'N U T, 0, 0, 0',
	X =  114.927  mm,	Y =   -296.118  mm,	Z =   -263.905  mm,
	W =  90.000 deg,	P =   0.000 deg,	R =   90.000 deg
};
P[581]{
   GP1:
	UF : 0, UT : 6,		CONFIG : 'N U T, 0, 0, 0',
	X =  114.226  mm,	Y =   -296.469  mm,	Z =   -263.577  mm,
	W =  90.000 deg,	P =   0.000 deg,	R =   90.000 deg
};
P[582]{
   GP1:
	UF : 0, UT : 6,		CONFIG : 'N U T, 0, 0, 0',
	X =  112.729  mm,	Y =   -297.317  mm,	Z =   -263.478  mm,
	W =  90.000 deg,	P =   0.000 deg,	R =   90.000 deg
};
P[583]{
   GP1:
	UF : 0, UT : 6,		CONFIG : 'N U T, 0, 0, 0',
	X =  112.064  mm,	Y =   -297.756  mm,	Z =   -263.808  mm,
	W =  90.000 deg,	P =   0.000 deg,	R =   90.000 deg
};
P[584]{
   GP1:
	UF : 0, UT : 6,		CONFIG : 'N U T, 0, 0, 0',
	X =  111.426  mm,	Y =   -298.123  mm,	Z =   -263.807  mm,
	W =  90.000 deg,	P =   0.000 deg,	R =   90.000 deg
};
P[585]{
   GP1:
	UF : 0, UT : 6,		CONFIG : 'N U T, 0, 0, 0',
	X =  109.718  mm,	Y =   -299.048  mm,	Z =   -263.431  mm,
	W =  90.000 deg,	P =   0.000 deg,	R =   90.000 deg
};
P[586]{
   GP1:
	UF : 0, UT : 6,		CONFIG : 'N U T, 0, 0, 0',
	X =  109.275  mm,	Y =   -299.370  mm,	Z =   -263.840  mm,
	W =  90.000 deg,	P =   0.000 deg,	R =   90.000 deg
};
P[587]{
   GP1:
	UF : 0, UT : 6,		CONFIG : 'N U T, 0, 0, 0',
	X =  107.984  mm,	Y =   -300.115  mm,	Z =   -263.831  mm,
	W =  90.000 deg,	P =   0.000 deg,	R =   90.000 deg
};
P[588]{
   GP1:
	UF : 0, UT : 6,		CONFIG : 'N U T, 0, 0, 0',
	X =  106.196  mm,	Y =   -301.115  mm,	Z =   -263.629  mm,
	W =  90.000 deg,	P =   0.000 deg,	R =   90.000 deg
};
P[589]{
   GP1:
	UF : 0, UT : 6,		CONFIG : 'N U T, 0, 0, 0',
	X =  105.606  mm,	Y =   -301.464  mm,	Z =   -263.680  mm,
	W =  90.000 deg,	P =   0.000 deg,	R =   90.000 deg
};
P[590]{
   GP1:
	UF : 0, UT : 6,		CONFIG : 'N U T, 0, 0, 0',
	X =  103.353  mm,	Y =   -302.801  mm,	Z =   -263.911  mm,
	W =  90.000 deg,	P =   0.000 deg,	R =   90.000 deg
};
P[591]{
   GP1:
	UF : 0, UT : 6,		CONFIG : 'N U T, 0, 0, 0',
	X =  100.868  mm,	Y =   -304.210  mm,	Z =   -263.749  mm,
	W =  90.000 deg,	P =   0.000 deg,	R =   90.000 deg
};
P[592]{
   GP1:
	UF : 0, UT : 6,		CONFIG : 'N U T, 0, 0, 0',
	X =  99.867  mm,	Y =   -304.780  mm,	Z =   -263.702  mm,
	W =  90.000 deg,	P =   0.000 deg,	R =   90.000 deg
};
P[593]{
   GP1:
	UF : 0, UT : 6,		CONFIG : 'N U T, 0, 0, 0',
	X =  99.162  mm,	Y =   -305.158  mm,	Z =   -263.520  mm,
	W =  90.000 deg,	P =   0.000 deg,	R =   90.000 deg
};
P[594]{
   GP1:
	UF : 0, UT : 6,		CONFIG : 'N U T, 0, 0, 0',
	X =  98.173  mm,	Y =   -305.730  mm,	Z =   -263.519  mm,
	W =  90.000 deg,	P =   0.000 deg,	R =   90.000 deg
};
P[595]{
   GP1:
	UF : 0, UT : 6,		CONFIG : 'N U T, 0, 0, 0',
	X =  96.024  mm,	Y =   -307.002  mm,	Z =   -263.718  mm,
	W =  90.000 deg,	P =   0.000 deg,	R =   90.000 deg
};
P[596]{
   GP1:
	UF : 0, UT : 6,		CONFIG : 'N U T, 0, 0, 0',
	X =  95.372  mm,	Y =   -307.392  mm,	Z =   -263.798  mm,
	W =  90.000 deg,	P =   0.000 deg,	R =   90.000 deg
};
P[597]{
   GP1:
	UF : 0, UT : 6,		CONFIG : 'N U T, 0, 0, 0',
	X =  93.908  mm,	Y =   -308.238  mm,	Z =   -263.802  mm,
	W =  90.000 deg,	P =   0.000 deg,	R =   90.000 deg
};
P[598]{
   GP1:
	UF : 0, UT : 6,		CONFIG : 'N U T, 0, 0, 0',
	X =  92.905  mm,	Y =   -308.781  mm,	Z =   -263.579  mm,
	W =  90.000 deg,	P =   0.000 deg,	R =   90.000 deg
};
P[599]{
   GP1:
	UF : 0, UT : 6,		CONFIG : 'N U T, 0, 0, 0',
	X =  91.246  mm,	Y =   -309.781  mm,	Z =   -263.845  mm,
	W =  90.000 deg,	P =   0.000 deg,	R =   90.000 deg
};
P[600]{
   GP1:
	UF : 0, UT : 6,		CONFIG : 'N U T, 0, 0, 0',
	X =  88.859  mm,	Y =   -311.165  mm,	Z =   -263.880  mm,
	W =  90.000 deg,	P =   0.000 deg,	R =   90.000 deg
};
P[601]{
   GP1:
	UF : 0, UT : 6,		CONFIG : 'N U T, 0, 0, 0',
	X =  87.677  mm,	Y =   -311.798  mm,	Z =   -263.575  mm,
	W =  90.000 deg,	P =   0.000 deg,	R =   90.000 deg
};
P[602]{
   GP1:
	UF : 0, UT : 6,		CONFIG : 'N U T, 0, 0, 0',
	X =  81.300  mm,	Y =   -315.516  mm,	Z =   -263.793  mm,
	W =  90.000 deg,	P =   0.000 deg,	R =   90.000 deg
};
P[603]{
   GP1:
	UF : 0, UT : 6,		CONFIG : 'N U T, 0, 0, 0',
	X =  80.189  mm,	Y =   -316.172  mm,	Z =   -263.881  mm,
	W =  90.000 deg,	P =   0.000 deg,	R =   90.000 deg
};
P[604]{
   GP1:
	UF : 0, UT : 6,		CONFIG : 'N U T, 0, 0, 0',
	X =  79.052  mm,	Y =   -316.764  mm,	Z =   -263.480  mm,
	W =  90.000 deg,	P =   0.000 deg,	R =   90.000 deg
};
P[605]{
   GP1:
	UF : 0, UT : 6,		CONFIG : 'N U T, 0, 0, 0',
	X =  78.460  mm,	Y =   -317.114  mm,	Z =   -263.535  mm,
	W =  90.000 deg,	P =   0.000 deg,	R =   90.000 deg
};
P[606]{
   GP1:
	UF : 0, UT : 6,		CONFIG : 'N U T, 0, 0, 0',
	X =  76.369  mm,	Y =   -318.360  mm,	Z =   -263.774  mm,
	W =  90.000 deg,	P =   0.000 deg,	R =   90.000 deg
};
P[607]{
   GP1:
	UF : 0, UT : 6,		CONFIG : 'N U T, 0, 0, 0',
	X =  74.036  mm,	Y =   -319.672  mm,	Z =   -263.561  mm,
	W =  90.000 deg,	P =   0.000 deg,	R =   90.000 deg
};
P[608]{
   GP1:
	UF : 0, UT : 6,		CONFIG : 'N U T, 0, 0, 0',
	X =  72.778  mm,	Y =   -320.443  mm,	Z =   -263.838  mm,
	W =  90.000 deg,	P =   0.000 deg,	R =   90.000 deg
};
P[609]{
   GP1:
	UF : 0, UT : 6,		CONFIG : 'N U T, 0, 0, 0',
	X =  70.664  mm,	Y =   -321.658  mm,	Z =   -263.796  mm,
	W =  90.000 deg,	P =   0.000 deg,	R =   90.000 deg
};
P[610]{
   GP1:
	UF : 0, UT : 6,		CONFIG : 'N U T, 0, 0, 0',
	X =  69.652  mm,	Y =   -322.194  mm,	Z =   -263.499  mm,
	W =  90.000 deg,	P =   0.000 deg,	R =   90.000 deg
};
P[611]{
   GP1:
	UF : 0, UT : 6,		CONFIG : 'N U T, 0, 0, 0',
	X =  68.123  mm,	Y =   -323.133  mm,	Z =   -263.850  mm,
	W =  90.000 deg,	P =   0.000 deg,	R =   90.000 deg
};
P[612]{
   GP1:
	UF : 0, UT : 6,		CONFIG : 'N U T, 0, 0, 0',
	X =  66.785  mm,	Y =   -323.887  mm,	Z =   -263.730  mm,
	W =  90.000 deg,	P =   0.000 deg,	R =   90.000 deg
};
P[613]{
   GP1:
	UF : 0, UT : 6,		CONFIG : 'N U T, 0, 0, 0',
	X =  65.868  mm,	Y =   -324.433  mm,	Z =   -263.838  mm,
	W =  90.000 deg,	P =   0.000 deg,	R =   90.000 deg
};
P[614]{
   GP1:
	UF : 0, UT : 6,		CONFIG : 'N U T, 0, 0, 0',
	X =  65.107  mm,	Y =   -324.873  mm,	Z =   -263.838  mm,
	W =  90.000 deg,	P =   0.000 deg,	R =   90.000 deg
};
P[615]{
   GP1:
	UF : 0, UT : 6,		CONFIG : 'N U T, 0, 0, 0',
	X =  64.287  mm,	Y =   -325.328  mm,	Z =   -263.725  mm,
	W =  90.000 deg,	P =   0.000 deg,	R =   90.000 deg
};
P[616]{
   GP1:
	UF : 0, UT : 6,		CONFIG : 'N U T, 0, 0, 0',
	X =  63.023  mm,	Y =   -326.040  mm,	Z =   -263.611  mm,
	W =  90.000 deg,	P =   0.000 deg,	R =   90.000 deg
};
P[617]{
   GP1:
	UF : 0, UT : 6,		CONFIG : 'N U T, 0, 0, 0',
	X =  62.107  mm,	Y =   -326.595  mm,	Z =   -263.776  mm,
	W =  90.000 deg,	P =   0.000 deg,	R =   90.000 deg
};
P[618]{
   GP1:
	UF : 0, UT : 6,		CONFIG : 'N U T, 0, 0, 0',
	X =  59.537  mm,	Y =   -328.096  mm,	Z =   -263.884  mm,
	W =  90.000 deg,	P =   0.000 deg,	R =   90.000 deg
};
P[619]{
   GP1:
	UF : 0, UT : 6,		CONFIG : 'N U T, 0, 0, 0',
	X =  57.711  mm,	Y =   -329.103  mm,	Z =   -263.587  mm,
	W =  90.000 deg,	P =   0.000 deg,	R =   90.000 deg
};
P[620]{
   GP1:
	UF : 0, UT : 6,		CONFIG : 'N U T, 0, 0, 0',
	X =  56.773  mm,	Y =   -329.618  mm,	Z =   -263.431  mm,
	W =  90.000 deg,	P =   0.000 deg,	R =   90.000 deg
};
P[621]{
   GP1:
	UF : 0, UT : 6,		CONFIG : 'N U T, 0, 0, 0',
	X =  56.142  mm,	Y =   -329.999  mm,	Z =   -263.525  mm,
	W =  90.000 deg,	P =   0.000 deg,	R =   90.000 deg
};
P[622]{
   GP1:
	UF : 0, UT : 6,		CONFIG : 'N U T, 0, 0, 0',
	X =  53.598  mm,	Y =   -330.475  mm,	Z =   -263.607  mm,
	W =  90.000 deg,	P =   0.000 deg,	R =   90.000 deg
};
P[623]{
   GP1:
	UF : 0, UT : 6,		CONFIG : 'N U T, 0, 0, 0',
	X =  54.713  mm,	Y =   -330.971  mm,	Z =   -263.777  mm,
	W =  90.000 deg,	P =   0.000 deg,	R =   90.000 deg
};
P[624]{
   GP1:
	UF : 0, UT : 6,		CONFIG : 'N U T, 0, 0, 0',
	X =  53.862  mm,	Y =   -331.942  mm,	Z =   -263.846  mm,
	W =  90.000 deg,	P =   0.000 deg,	R =   90.000 deg
};
P[625]{
   GP1:
	UF : 0, UT : 6,		CONFIG : 'N U T, 0, 0, 0',
	X =  52.588  mm,	Y =   -331.620  mm,	Z =   -263.902  mm,
	W =  90.000 deg,	P =   0.000 deg,	R =   90.000 deg
};
P[626]{
   GP1:
	UF : 0, UT : 6,		CONFIG : 'N U T, 0, 0, 0',
	X =  52.240  mm,	Y =   -332.373  mm,	Z =   -263.888  mm,
	W =  90.000 deg,	P =   0.000 deg,	R =   90.000 deg
};
P[627]{
   GP1:
	UF : 0, UT : 6,		CONFIG : 'N U T, 0, 0, 0',
	X =  53.428  mm,	Y =   -332.974  mm,	Z =   -263.876  mm,
	W =  90.000 deg,	P =   0.000 deg,	R =   90.000 deg
};
P[628]{
   GP1:
	UF : 0, UT : 6,		CONFIG : 'N U T, 0, 0, 0',
	X =  52.003  mm,	Y =   -333.365  mm,	Z =   -263.813  mm,
	W =  90.000 deg,	P =   0.000 deg,	R =   90.000 deg
};
P[629]{
   GP1:
	UF : 0, UT : 6,		CONFIG : 'N U T, 0, 0, 0',
	X =  53.574  mm,	Y =   -335.798  mm,	Z =   -263.468  mm,
	W =  90.000 deg,	P =   0.000 deg,	R =   90.000 deg
};
P[630]{
   GP1:
	UF : 0, UT : 6,		CONFIG : 'N U T, 0, 0, 0',
	X =  52.426  mm,	Y =   -335.739  mm,	Z =   -263.524  mm,
	W =  90.000 deg,	P =   0.000 deg,	R =   90.000 deg
};
P[631]{
   GP1:
	UF : 0, UT : 6,		CONFIG : 'N U T, 0, 0, 0',
	X =  54.582  mm,	Y =   -337.530  mm,	Z =   -263.866  mm,
	W =  90.000 deg,	P =   0.000 deg,	R =   90.000 deg
};
P[632]{
   GP1:
	UF : 0, UT : 6,		CONFIG : 'N U T, 0, 0, 0',
	X =  55.071  mm,	Y =   -338.463  mm,	Z =   -263.563  mm,
	W =  90.000 deg,	P =   0.000 deg,	R =   90.000 deg
};
P[633]{
   GP1:
	UF : 0, UT : 6,		CONFIG : 'N U T, 0, 0, 0',
	X =  55.596  mm,	Y =   -339.307  mm,	Z =   -263.791  mm,
	W =  90.000 deg,	P =   0.000 deg,	R =   90.000 deg
};
P[634]{
   GP1:
	UF : 0, UT : 6,		CONFIG : 'N U T, 0, 0, 0',
	X =  57.256  mm,	Y =   -342.183  mm,	Z =   -263.786  mm,
	W =  90.000 deg,	P =   0.000 deg,	R =   90.000 deg
};
P[635]{
   GP1:
	UF : 0, UT : 6,		CONFIG : 'N U T, 0, 0, 0',
	X =  58.086  mm,	Y =   -343.621  mm,	Z =   -263.781  mm,
	W =  90.000 deg,	P =   0.000 deg,	R =   90.000 deg
};
P[636]{
   GP1:
	UF : 0, UT : 6,		CONFIG : 'N U T, 0, 0, 0',
	X =  58.492  mm,	Y =   -344.293  mm,	Z =   -263.898  mm,
	W =  90.000 deg,	P =   0.000 deg,	R =   90.000 deg
};
P[637]{
   GP1:
	UF : 0, UT : 6,		CONFIG : 'N U T, 0, 0, 0',
	X =  59.378  mm,	Y =   -345.910  mm,	Z =   -263.596  mm,
	W =  90.000 deg,	P =   0.000 deg,	R =   90.000 deg
};
P[638]{
   GP1:
	UF : 0, UT : 6,		CONFIG : 'N U T, 0, 0, 0',
	X =  60.035  mm,	Y =   -347.032  mm,	Z =   -263.658  mm,
	W =  90.000 deg,	P =   0.000 deg,	R =   90.000 deg
};
P[639]{
   GP1:
	UF : 0, UT : 6,		CONFIG : 'N U T, 0, 0, 0',
	X =  60.894  mm,	Y =   -348.513  mm,	Z =   -263.676  mm,
	W =  90.000 deg,	P =   0.000 deg,	R =   90.000 deg
};
P[640]{
   GP1:
	UF : 0, UT : 6,		CONFIG : 'N U T, 0, 0, 0',
	X =  61.275  mm,	Y =   -349.176  mm,	Z =   -263.670  mm,
	W =  90.000 deg,	P =   0.000 deg,	R =   90.000 deg
};
P[641]{
   GP1:
	UF : 0, UT : 6,		CONFIG : 'N U T, 0, 0, 0',
	X =  61.838  mm,	Y =   -350.182  mm,	Z =   -263.561  mm,
	W =  90.000 deg,	P =   0.000 deg,	R =   90.000 deg
};
P[642]{
   GP1:
	UF : 0, UT : 6,		CONFIG : 'N U T, 0, 0, 0',
	X =  62.286  mm,	Y =   -350.994  mm,	Z =   -263.429  mm,
	W =  90.000 deg,	P =   0.000 deg,	R =   90.000 deg
};
P[643]{
   GP1:
	UF : 0, UT : 6,		CONFIG : 'N U T, 0, 0, 0',
	X =  63.009  mm,	Y =   -352.130  mm,	Z =   -263.842  mm,
	W =  90.000 deg,	P =   0.000 deg,	R =   90.000 deg
};
P[644]{
   GP1:
	UF : 0, UT : 6,		CONFIG : 'N U T, 0, 0, 0',
	X =  63.417  mm,	Y =   -352.948  mm,	Z =   -263.446  mm,
	W =  90.000 deg,	P =   0.000 deg,	R =   90.000 deg
};
P[645]{
   GP1:
	UF : 0, UT : 6,		CONFIG : 'N U T, 0, 0, 0',
	X =  63.975  mm,	Y =   -353.810  mm,	Z =   -263.819  mm,
	W =  90.000 deg,	P =   0.000 deg,	R =   90.000 deg
};
P[646]{
   GP1:
	UF : 0, UT : 6,		CONFIG : 'N U T, 0, 0, 0',
	X =  64.727  mm,	Y =   -355.216  mm,	Z =   -263.451  mm,
	W =  90.000 deg,	P =   0.000 deg,	R =   90.000 deg
};
P[647]{
   GP1:
	UF : 0, UT : 6,		CONFIG : 'N U T, 0, 0, 0',
	X =  65.308  mm,	Y =   -356.137  mm,	Z =   -263.757  mm,
	W =  90.000 deg,	P =   0.000 deg,	R =   90.000 deg
};
P[648]{
   GP1:
	UF : 0, UT : 6,		CONFIG : 'N U T, 0, 0, 0',
	X =  66.017  mm,	Y =   -357.348  mm,	Z =   -263.818  mm,
	W =  90.000 deg,	P =   0.000 deg,	R =   90.000 deg
};
P[649]{
   GP1:
	UF : 0, UT : 6,		CONFIG : 'N U T, 0, 0, 0',
	X =  66.559  mm,	Y =   -358.380  mm,	Z =   -263.482  mm,
	W =  90.000 deg,	P =   0.000 deg,	R =   90.000 deg
};
P[650]{
   GP1:
	UF : 0, UT : 6,		CONFIG : 'N U T, 0, 0, 0',
	X =  67.615  mm,	Y =   -360.190  mm,	Z =   -263.546  mm,
	W =  90.000 deg,	P =   0.000 deg,	R =   90.000 deg
};
P[651]{
   GP1:
	UF : 0, UT : 6,		CONFIG : 'N U T, 0, 0, 0',
	X =  68.727  mm,	Y =   -362.046  mm,	Z =   -263.800  mm,
	W =  90.000 deg,	P =   0.000 deg,	R =   90.000 deg
};
P[652]{
   GP1:
	UF : 0, UT : 6,		CONFIG : 'N U T, 0, 0, 0',
	X =  69.449  mm,	Y =   -363.296  mm,	Z =   -263.798  mm,
	W =  90.000 deg,	P =   0.000 deg,	R =   90.000 deg
};
P[653]{
   GP1:
	UF : 0, UT : 6,		CONFIG : 'N U T, 0, 0, 0',
